    INIT := 100, // Initialisieren 
    Init_HomeVertical_10,
    Init_Vertical_10_Down,
    Init_HomeVertical_02,
    Init_Vertical_02_Up,
    Init_HomeHorizontal,
    Init_HorizontalToTrack,
    Init_check_if_pces_handled,

    READY := 999,  // READY to Start, Init Done 
    START := 1000, // Start Zyklisch

    waitOnMover,     // wait until the mover is there
    MOVER_NEEDED_OP, // Ab here, a mover in position is needed to perform the action

    lift_piece_and_down_to_pick,        // lift the piece with 180.10Z and go down simultaneously with 180.02Z
    close_griper_pick_piece,            // close the griper to pick the piece
    clamp_down_maintain_piece,          // the clamp (niederhalter) goes down and hold the piece in place
    take_out_piece_and_put_down_lifter, // 180.02Z goes up with the piece, 180.10Z goes down

    SYNC_MOVER_LEAVE, // MoverMan need to take the mover
    MOVER_FREE_OP,    // here, operation without mover can be done.

    hor_move_to_extraction_pipe, // 180.01Y move to the extraction pipe
    ver_down_in_pipe,            // 180.02Z move down to a secure position to release the piece
    open_griper_put_piece,
    clamp_up_to_rest_position,
    ver_up_empty, // 180.02z goes up without piece
    hor_to_track_pos,
    ver_down_waiting_for_mover, // go down again and wait until a mover is there

    DONE := 8000,  // Ablauf beendet 
    ERROR := 9000, // Fehler 
    _max
);
END_TYPE

(*
back to shuttle
check level NIO Box
*)

// ---- POUs/20_AUTO/ST180/ST180_Recipe_t.TcDUT
TYPE ST180_Recipe_t : 
STRUCT
    xUseVerLeft  : BOOL; // Is the left vertical picker element is used
    xUseVerRight : BOOL; // Is the right vertical picker element is used
END_STRUCT
END_TYPE

// ---- POUs/20_AUTO/ST185/ST185_Cylinders_e.TcTLEO
TYPE ST185_Cylinders_e :
(
    Greifer_Patrone_Links,
    Greifer_Patrone_Rechts,
    Niederhalter_Deckel_Links,
    Niederhalter_Deckel_Rechts
);
END_TYPE

// ---- POUs/20_AUTO/ST185/ST185_PnpHorPos_e.TcDUT
TYPE ST185_PnpHorPos_e : ST110_PnpHorPos_e;
END_TYPE

// ---- POUs/20_AUTO/ST185/ST185_PnpVerPos_e.TcDUT
TYPE ST185_PnpVerPos_e :
(
    up_waiting_mover,
    down_empty,
    up_full,
    down_full,
	up_after_unload,
    _max
);
END_TYPE

// ---- POUs/20_AUTO/ST185/ST185_Pnp_e.TcTLEO
{attribute 'qualified_only'}
{attribute 'strict'}
{attribute 'to_string'}
TYPE
ST185_Pnp_e :
(
    RESET := 0, // Reset

    INIT := 100, // Initialisieren 
    Init_HomeVertical_10,
    Init_Vertical_10_Down,
    Init_HomeVertical_02,
    Init_Vertical_02_Up,
    Init_HomeHorizontal,
    Init_HorizontalToTrack,
    Init_check_if_pces_handled,

    READY := 999,  // READY to Start, Init Done 
    START := 1000, // Start Zyklisch

    waitOnMover,     // wait until the mover is there
    MOVER_NEEDED_OP, // Ab here, a mover in position is needed to perform the action

    lift_piece_and_down_to_pick,        // lift the piece with 180.10Z and go down simultaneously with 180.02Z
    close_griper_pick_piece,            // close the griper to pick the piece
    clamp_down_maintain_piece,          // the clamp (niederhalter) goes down and hold the piece in place
    take_out_piece_and_put_down_lifter, // 180.02Z goes up with the piece, 180.10Z goes down

    SYNC_MOVER_LEAVE, // MoverMan need to take the mover
    MOVER_FREE_OP,    // here, operation without mover can be done.

    hor_move_to_extraction_pipe, // 180.01Y move to the extraction pipe
    ver_down_in_pipe,            // 180.02Z move down to a secure position to release the piece
    open_griper_put_piece,
    clamp_up_to_rest_position,
    ver_up_empty, // 180.02z goes up without piece
    hor_to_track_pos,
    ver_down_waiting_for_mover, // go down again and wait until a mover is there

    DONE := 8000,  // Ablauf beendet 
    ERROR := 9000, // Fehler 
    _max
);
END_TYPE

(*
back to shuttle
check level NIO Box
*)

// ---- POUs/20_AUTO/ST185/ST185_Recipe_t.TcDUT
TYPE ST185_Recipe_t : 
STRUCT
    xUseVerLeft  : BOOL; // Is the left vertical picker element is used
    xUseVerRight : BOOL; // Is the right vertical picker element is used
END_STRUCT
END_TYPE

// ---- POUs/20_AUTO/StationList_e.TcTLEO
// Only station with manual mode cylinders
{attribute 'qualified_only'}
TYPE StationList_e :
(
    ST105, // 0
    ST110, // 1
    ST115, // 2
    ST120, // 3
    ST125, // 4
    ST128, // 5
    ST130, // 6
    ST135, // 7
    ST140, // 8
    ST145, // 9
    ST150, // 10
    ST155, // 11
    ST160, // 12
    ST165, // 13
    ST170, // 14
    //ST174 // is ignored because it is a waiting station
    ST175, // 15
    ST176, // 16
    ST180, // 17
    ST185, // 18
	_max
);
END_TYPE

// ---- GVLs/AXIS.TcGVL
{attribute 'qualified_only'}
(*******************************************************************)
(* ACHSEN KONSTANTEN *)
(*******************************************************************)
VAR_GLOBAL CONSTANT

END_VAR
VAR_GLOBAL
    (*******************************************************************)
    (* ACHSEN Variablen *)
    (*******************************************************************)
    //Axis Allgemein Teachen und Anzeige
    bTeachAxisNr  : BYTE;                              // Zu Teachende Achse # (von HMI)
    bTeachInPos   : BYTE;                              // Achse in Position (Teachpos (99= nicht in Pos))
    bTeachPos     : ARRAY[0..Axis_e._max - 1] OF BYTE; // Achse Teach Position (Anzufahrende Position #)
    rTeachIncAxis : REAL := 0.1;                       // Axis Inching Wert
    rTeachVelo    : REAL := 10;                        // Achse Geschwindigkeit (Anzeige)
    rTeachPos     : REAL;                              // Achse Teach Position (Anzufahrende Position Wert)
    rTeachActPos  : REAL;                              // Achse AKTUELLE Position (AKTUEL
    rTeachPosMin  : REAL;                              // Achse PositionsminimumLER Position Wert)
    rTeachPosMax  : REAL;                              // Achse Positionsmaximum
    rJogVelo_pc   : REAL := REAL#10.0;                 // global jog velocity in pc

    btTeachArAxis : ARRAY[0..Axis_e._max - 1] OF ARRAY[0..8] OF structButton; (* Buttons AXIS
                                                    0: Disable 
                                                    1: Inching 
                                                    2: Slow 
                                                    3: Fast 
                                                    4: Move Abs/Rel   
                                                    5: Manu Move NEGATIVE
                                                    6: Manu Move POSITIVE  
													7: Start Homing 
													8: Teachpos Übernehmen*)
END_VAR

(*******************************************************************)
(* ACHSEN Positionen von HMI*)
(*******************************************************************)
VAR_GLOBAL RETAIN

END_VAR

// ---- GVLs/CONST.TcGVL
{attribute 'qualified_only' := ''}
VAR_GLOBAL CONSTANT
    (*******************************************************************)
    (* Globale KONSTANTEN *)
    (*******************************************************************)

    USE_SIMULATION  : BOOL := TRUE;
    BIND_WITH_TRACK : BOOL := TRUE;

    STATION_NUMBER           : INT   := 20;
    MAX_GROUP                : INT   := 6;
    MAX_STATION_PER_GROUP    : INT   := 8;
    MAX_RECIPE_NUMBER        : INT   := 11;
    MAX_TRACK_LENGTH         : LREAL := 10060;
    MAX_MOVER_SIZE           : LREAL := 200.0;
    MAX_VECTOR_LIST          : INT   := 10;
    MAX_CYLINDER_PER_STATION : INT   := 10;

END_VAR

// ---- GVLs/GVL.TcGVL
{attribute 'qualified_only'}
VAR_GLOBAL
    (*******************************************************************)
    (* Allgemeine Globale Variablen *)
    (*******************************************************************)
    (******* FREIGABEN *********)
    //ST01
    xFG_ST01akVZ : BOOL; // Vereinzelung Teil anwesend
    xFG_ST01akWT : BOOL; // WT anwesend
    //ST02
    xFG_ST02akWT : BOOL; // WT anwesend

    st105_aut : FB_AUT_105;    // Laden Filtergehäuse
    st110_aut : FB_AUT_110;    // Laden RFID-Ring
    st115_aut : FB_AUT_115;    // Laden kristal
    st120_aut : FB_AUT_120;    // Laden Solerohr
    st125_aut : FB_AUT_125;    // Laden filterhut
    st128_aut : FB_AUT_128;    // Control filterhut
    st130_aut : FB_AUT_130;    // Dosieren A
    st135_aut : FB_AUT_135;    // Dosieren B
    st140_aut : FB_AUT_140;    // Niveaukontrolle
    st145_aut : FB_AUT_145;    // Laden Patronendeckel
    st150_aut : FB_AUT_150;    // Utralson A
    st155_aut : FB_AUT_155;    // Ultrason B
    st160_aut : FB_AUT_160;    // Prüfig A
    st165_aut : FB_AUT_165;    // Prüfig B
    st170_aut : FB_AUT_170;    // Program RFID
    st175_aut : FB_AUT_175;    // Laser A
    st176_aut : FB_AUT_MODIFY; // Laser B
    st180_aut : FB_AUT_180;    // Entladen schlecht
    st185_aut : FB_AUT_185;    // Entladen gut
	
	ST130_01Y_Feedback_Offset : LREAL; // Offset automatically adjusted by ST140
	ST135_01Y_Feedback_Offset : LREAL; // Offset automatically adjusted by ST140

END_VAR

// ---- GVLs/HMI.TcGVL
{attribute 'qualified_only'}
VAR_GLOBAL
    (*******************************************************************)
    (* Globale HMI Variablen *)
    (*******************************************************************)
    xImmer0 : BOOL := FALSE; //ALLWAYS FALSE
    xImmer1 : BOOL := TRUE;  //ALLWAYS TRUE

    (*******************************************************************)
    (* Flags *)
    (*******************************************************************)
    enState   : enState; //SYSTEM STATUS
    xInitDone : BOOL;    //SYSTEM INITIALIZED
    xRefDone  : BOOL;    //Axis REF
    xAlarm    : BOOL;    //ALARM AKTIV
    xMessage  : BOOL;    //MELDUNG AKTIV
    xWait     : BOOL;    //ALLE FBs warten
    xAIRon    : BOOL;    //Luftdruck IO
    xSPC      : BOOL;    //SPC angewählt

    Tast_BL : BOOL; // ... 

    (*******************************************************************)
    (* Buttons *)
    (*******************************************************************)
    //Control
    btArMain : ARRAY[0..20] OF structButton; (*	
													0: AUTO
													1: STEP
													2: END
													3: MANU
													4: INIT
													5: STOP
													6: LEER
													7: QUIT
													8: RESET TEMP COUNTER
													9: START
													10: HUBTÜREn ALLE
													11: HUBTÜRE 1
													12: HUBTÜRE 2
													13: HUBTÜRE 3
													14: HUBTÜRE 4
												*)
    //Manual pneumatics
    // see below for button button instance 
    btManuCylinders : ARRAY[0..StationList_e._max] OF ARRAY[0..CONST.MAX_CYLINDER_PER_STATION] OF structButton;
    (* 
	 * [StationList_e.ST105] 0
     * [0]: Zyklus [1]: Robot get [2]: Robot set [3] Feeder
	 *
     * [StationList_e.ST110] 1
     * [0]: Zyklus [1]: Vacum Gripper left [2]: Vacum Gripper right [3]: Feeder
     *
     * [StationList_e.ST115] 2
     * [0]: Zyklus [1]: Gripper left [2]: Gripper right [3]: Feeder
     *
     * [StationList_e.ST120] 3
     * [0]: Zyklus [1]: Gripper left [2]: Gripper right [3]: Rotative cylinder left
     * [4]: Rotative cylinder right [5]: Hublader left [6]: Hublader right
	 * [7]: feeder left [8]: feeder right
     *
     * [StationList_e.ST125] 4
     * [0]: Zyklus [1]: Gripper left [2]: Gripper right [3]: lock cylinder left
     * [4]: lock cylinder right [5]: Gripper Solerohr left [6]: Gripper Solerohr right
	 * [7]: feeder 
     *
     * [StationList_e.ST130] 5
     * [0]: Zyklus [1]: cell open left [2]: cell open right [3]: cell fill left
     * [4]: cell fill right [5]: vib cell left [6]: vib cell right
	 * [7]: holder patrone [8]: vib patrone left [9]: vib patrone right [10]: Feeder 
     *
     * [StationList_e.ST135] 6
	 * dito ST130
	 *
     * [StationList_e.ST145] 8
     * [0]: Zyklus [1]: Vacum Gripper left [2]: Vacum Gripper right [3]: Feeder
	 *
     * [StationList_e.ST150] 9
     * [0]: Zyklus [1]: mover maintening [2]: start welding
	 *
     * [StationList_e.ST155] 10
     * [0]: Zyklus [1]: mover maintening [2]: start welding
	 *
     * [StationList_e.ST160] 11
     * [0]: Zyklus [1]: holder left [2]: holder right [3]: seal left
	 * [4]: seal right [5]: fill left [6]: fill right [7]: start test
	 *
     * [StationList_e.ST165] 12
     * [0]: Zyklus [1]: holder left [2]: holder right [3]: seal left
	 * [4]: seal right [5]: fill left [6]: fill right [7]: start test
	 *
     * [StationList_e.ST170] 13
     * [0]: Zyklus [1]: start test left [2]: start test right
	 *
     * [StationList_e.ST175] 14
     * [0]: Zyklus [1]: holder [2]: cabine in [3]: cabine out
	 * [4]: start laser
	 *
     * [StationList_e.ST180] 15
     * [0]: Zyklus [1]: Gripper left [2]: Gripper right 
	 * [3]: holder left [4]: holder right
	 *
     * [StationList_e.ST185] 11
     * [0]: Zyklus [1]:  [2]: 
     *)

    btArST150 : ARRAY[0..20] OF structButton; (*	0 : Start USS
	                                                1 : Reset US
											   *)

    btArForceCyclus     : ARRAY[0..StationList_e._max - 1] OF structButton;
    bArForceCyclusState : ARRAY[0..StationList_e._max - 1] OF BOOL;

    (*******************************************************************)
    (* ALARME  *)
    (*******************************************************************)
    strArALARM  : ARRAY[1..100] OF structAlarm;
    strArMSG    : ARRAY[1..100] OF structAlarm;
    xArAlarmHMI : ARRAY[1..9999] OF BOOL;

    (*******************************************************************)
    (* ANZEIGE - Werte *)
    (*******************************************************************)
    iSelectAxis     : LinearAxis_e := LinearAxis_e.ST110_01Y;
    iSelectAxisCopy : LinearAxis_e := LinearAxis_e._max;
    btCopyAxisCfg   : structButton;

    iSelectCylinder     : StationList_e := StationList_e.ST105;
    iSelectCylinderCopy : StationList_e := StationList_e._max;
    btCopyCylinderCfg   : structButton;

    iSelectJogAxis : Axis_e;

    (*******************************************************************)
    (* Cycle Time [STATION]*)
    (*******************************************************************)
    dwArStartTime_ms : ARRAY[0..StationList_e._max - 1] OF DWORD;
    dwArCycleTime_ms : ARRAY[0..StationList_e._max - 1] OF DWORD;

    lrPiecePerMinute : LREAL;

    PieceDoneTmp : DINT; // number of piece done since last reset

    (*******************************************************************)
    (* Recipe HMI management *)
    (*******************************************************************)
    btCopyRecipe  : structButton;
    btSetDefault  : structButton;
    movesNames    : ARRAY[0..LinearAxis_e._max - 1] OF ARRAY[0..CONST.MAX_VECTOR_LIST] OF STRING;
    cylinderNames : ARRAY[0..StationList_e._max - 1] OF ARRAY[0..CONST.MAX_CYLINDER_PER_STATION] OF STRING;

    (*******************************************************************)
    (* Mover manual bt *)
    (*******************************************************************)
    selectedShuttle : INT := 1; // selected shuttle from the HMI

    (*******************************************************************)
    (* Diverses *)
    (*******************************************************************)
    xWriteALlog : BOOL;         // Alarmlog schreiben in File
    btWritePers : structButton; // write pers data in filesystem

    sCurrentHMI2 : STRING; // ???
END_VAR

// ---- GVLs/IN.TcGVL
{attribute 'qualified_only'}
VAR_GLOBAL
    (*******************************************************************)
    (* EINGÄNGE Schrank A *)
    (*******************************************************************)
    (* Modul *)
    //-EL1809 16DI 155D2
    I000_                          AT %IX00.0 : BOOL; //
    I001_monitor_24V               AT %IX00.1 : BOOL; // Netzgerät Schaltschrank A Überwachung +24V
    I002_monitor_BR                AT %IX00.2 : BOOL; // Netzgerüt B&R Überwachung +24V
    I003_lufter_safety             AT %IX00.3 : BOOL; // Lüfter Safety ok
    I004_druckwachter_luftdruck_ok AT %IX00.4 : BOOL; // Druckwächter Luftdruck ok
    I005_klimagerat_ok             AT %IX00.5 : BOOL; // Klimagerät ok
    I006_                          AT %IX00.6 : BOOL; //
    I007_                          AT %IX00.7 : BOOL; //

    I010_distanzsensor_verschmutzung_140_51 AT %IX01.0 : BOOL; // Distanzsensor 140.51 Verschmutzung
    I011_distanzsensor_verschmutzung_140_52 AT %IX01.1 : BOOL; // Distanzsensor 140.52 Verschmutzung
    I012_                                   AT %IX01.2 : BOOL; // 
    I013_                                   AT %IX01.3 : BOOL; // 
    I014_                                   AT %IX01.4 : BOOL; // 
    I015_                                   AT %IX01.5 : BOOL; // 
    I016_                                   AT %IX01.6 : BOOL; // 
    I017_                                   AT %IX01.7 : BOOL; // 

    //-EL1809 16DI 155D7
    I020_ultraschall_bereit_150_20  AT %IX02.0 : BOOL; // Ultraschall 150.20 Bereit
    I021_ultraschall_fehler_150_20  AT %IX02.1 : BOOL; // Ultraschall 150.20 Fehler
    I022_ultraschall_us_on_150_20   AT %IX02.2 : BOOL; // Ultraschall 150.20 US on
    I023_ultraschall_nullpos_150_20 AT %IX02.3 : BOOL; // Ultraschall 150.20 Nullposition
    I024_ultraschall_bereit_155_20  AT %IX02.4 : BOOL; // Ultraschall 155.20 Bereit
    I025_ultraschall_fehler_155_20  AT %IX02.5 : BOOL; // Ultraschall 155.20 Fehler
    I026_ultraschall_us_on_155_20   AT %IX02.6 : BOOL; // Ultraschall 155.20 US on
    I027_ultraschall_nullpos_155_20 AT %IX02.7 : BOOL; // Ultraschall 155.20 Nullposifion

    I030_rfid_test_link_out1_170_20 AT %IX03.0 : BOOL; // RFID Test links 170.20 OUT 1
    I031_rfid_test_link_out2_170_20 AT %IX03.1 : BOOL; // RFID Test links 170.20 OUT 2
    I032_rfid_test_link_out3_170_20 AT %IX03.2 : BOOL; // RFID Test links 170.20 OUT 3
    I033_rfid_test_link_out1_170_21 AT %IX03.3 : BOOL; // RFID Test links 170.21 OUT 1
    I034_rfid_test_link_out2_170_21 AT %IX03.4 : BOOL; // RFID Test links 170.21 OUT 2
    I035_rfid_test_link_out3_170_21 AT %IX03.5 : BOOL; // RFID Test links 170.21 OUT 3
    I036_                           AT %IX03.6 : BOOL; // 
    I037_                           AT %IX03.7 : BOOL; // 

    //-EL1809 16DI 15602
    I040_ AT %IX04.0 : BOOL; // 
    I041_ AT %IX04.1 : BOOL; // 
    I042_ AT %IX04.2 : BOOL; // 
    I043_ AT %IX04.3 : BOOL; // 
    I044_ AT %IX04.4 : BOOL; // 
    I045_ AT %IX04.5 : BOOL; // 
    I046_ AT %IX04.6 : BOOL; // 
    I047_ AT %IX04.7 : BOOL; // 

    I050_ AT %IX05.0 : BOOL; // 
    I051_ AT %IX05.1 : BOOL; // 
    I052_ AT %IX05.2 : BOOL; // 
    I053_ AT %IX05.3 : BOOL; // 
    I054_ AT %IX05.4 : BOOL; // 
    I055_ AT %IX05.5 : BOOL; // 
    I056_ AT %IX05.6 : BOOL; // 
    I057_ AT %IX05.7 : BOOL; // 

    (*******************************************************************)
    (* EINGÄNGE Schrank B *)
    (*******************************************************************)
    (* Modul *)
    //-EL1809 16DI 10155D2
    I500_laser_sammelfehler_175          AT %IX50.0 : BOOL; // Sauger Laser 175.21 Sammelfehler
    I501_laser_filter_voll_175           AT %IX50.1 : BOOL; // Sauger Laser 175.21 Filter voll
    I502_laser_drehzahl_175              AT %IX50.2 : BOOL; // Sauger Laser 175.21 Drehzahl
    I503_laser_temperatur_175            AT %IX50.3 : BOOL; // Sauger Laser 175.21 Temperatur
    I504_distanzsensor_verschmutzung_125 AT %IX50.4 : BOOL; // Distanzsensor 125.51 Verschmutzung
    I505_uberwachung_24V                 AT %IX50.5 : BOOL; // Netzgerät Schaltschrank B Überwachung +24V
    I506_klimagerat_ok                   AT %IX50.6 : BOOL; // Klimagerät schaltschrank B ok
    I507_entladeBand_125_alarm           AT %IX50.7 : BOOL; // Entladeband 185.21 Alarm

    I510_lufter_safey_ok AT %IX51.0 : BOOL; // Lüfter Safety Schaltschrank B ok
    I511_                AT %IX51.1 : BOOL; // 
    I512_                AT %IX51.2 : BOOL; // 
    I513_                AT %IX51.3 : BOOL; // 
    I514_                AT %IX51.4 : BOOL; // 
    I515_                AT %IX51.5 : BOOL; // 
    I516_                AT %IX51.6 : BOOL; // 
    I517_                AT %IX51.7 : BOOL; // 

    //-EL1809 16DI 1015507
    I520_                AT %IX52.0 : BOOL; // 
    I521_ AT %IX52.1 : BOOL; // 
    I522_                AT %IX52.2 : BOOL; // 
    I523_ AT %IX52.3 : BOOL; // 
    I524_                AT %IX52.4 : BOOL; // 
    I525_ AT %IX52.5 : BOOL; // 
    I526_                AT %IX52.6 : BOOL; // 
    I527_ AT %IX52.7 : BOOL; // 

    I530_ AT %IX53.0 : BOOL; // 
    I531_ AT %IX53.1 : BOOL; // 
    I532_ AT %IX53.2 : BOOL; // 
    I533_ AT %IX53.3 : BOOL; // 
    I534_ AT %IX53.4 : BOOL; // 
    I535_ AT %IX53.5 : BOOL; // 
    I536_ AT %IX53.6 : BOOL; // 
    I537_ AT %IX53.7 : BOOL; // 

    AI01_ST140_level_track_side AT %I* : UINT; // laser sensor used to measure powder level, placed at the track side
    AI02_ST140_level_door_side  AT %I* : UINT; // laser sensor used to measure powder level, placed at the door side

    AI11_ST130_valve_feedback_left  AT %I* : UINT; // current flow of the proportional valve
    AI12_ST130_valve_feedback_right AT %I* : UINT; // current flow of the proportional valve
    AI13_ST135_valve_feedback_left  AT %I* : UINT; // current flow of the proportional valve
    AI14_ST135_valve_feedback_right AT %I* : UINT; // current flow of the proportional valve

    AI21_ST125_piece_height AT %I* : UINT; // laser sensor value, detect pieces in round table
    AI22_                   AT %I* : UINT;

    I_CPX9_1_ResetBp AT %I* : BOOL; // Blue button on the panel
    I_CPX9_1_greenBp AT %I* : BOOL; // Green button on the panel
    I_CPX9_1_redBp   AT %I* : BOOL; // Red button on the panel

END_VAR

// ---- GVLs/IO_BOX.TcGVL
{attribute 'qualified_only'}
VAR_GLOBAL
    (*******************************************************************)
    (* EINGÄNGE Schrank A *)
    (*******************************************************************)

    (* IO-Link Boxen 190A1 *)
    (*******************************************************************)
    //-194A3
    (* BN Lampe *)
    I0000_ AT %Q* : BOOL; // lampe

    //-201A1
    (* Ventil Batterie 201 A*)
    Q0100_14_ST130_kammer_offnen_links     AT %Q* : BOOL; // ST130 Kammer öffnen links
    Q0100_12_                              AT %Q* : BOOL; // 
    Q0101_14_ST130_kammer_offnen_rechts     AT %Q* : BOOL; // ST130 Kammer öffnen rechts
    Q0101_12_                              AT %Q* : BOOL; // 
    Q0102_14_ST130_kammer_nachfullen_links  AT %Q* : BOOL; // ST130 Kammer nachfüllen links
    Q0102_12_                              AT %Q* : BOOL; // 
    Q0103_14_ST130_kammer_nachfullen_rechts AT %Q* : BOOL; // ST130 Kammer nachfüllen rechts
    Q0103_12_                              AT %Q* : BOOL; // 
    Q0104_14_ST130_vibrieren_kammer_links   AT %Q* : BOOL; // ST130 Vibrieren Kammer links/rechts aus
    Q0104_12_ST130_vibrieren_kammer_rechts AT %Q* : BOOL; // ST130 Vibrieren Kammer links/rechts ein
    Q0105_14_ST130_niederhalter_patrone    AT %Q* : BOOL; // ST130 Niederhalter Patrone
    Q0105_12_                              AT %Q* : BOOL; // 
    Q0106_14_ST135_kammer_offnen_links      AT %Q* : BOOL; // ST135 Kammer öffnen links
    Q0106_12_                              AT %Q* : BOOL; // 
    Q0107_14_ST135_kammer_offnen_rechts     AT %Q* : BOOL; // ST135 Kammer öffnen rechts
    Q0107_12_                              AT %Q* : BOOL; // 
    Q0108_14_ST135_kammer_nachfullen_links  AT %Q* : BOOL; // ST135 Kammer nachfüllen links
    Q0108_12_                              AT %Q* : BOOL; // 
    Q0109_14_ST135_kammer_nachfullen_rechts AT %Q* : BOOL; // ST135 Kammer nachfüllen rechts
    Q0109_12_                              AT %Q* : BOOL; // 
    Q0110_14_ST135_vibrieren_kammer_links   AT %Q* : BOOL; // ST135 Vibrieren Kammer links 
    Q0110_12_ST135_vibrieren_kammer_rechts AT %Q* : BOOL; // ST135 Vibrieren Kammer rechts
    Q0111_14_ST135_niederhalter_patrone    AT %Q* : BOOL; // ST135 Niederhalter Patrone
    Q0111_12                               AT %Q* : BOOL; //
    Q0112_14_                               AT %Q* : BOOL; //
    Q0112_12_                              AT %Q* : BOOL; // 
    Q0113_14_                               AT %Q* : BOOL; //
    Q0113_12_                              AT %Q* : BOOL; // 
    Q0114_14_                               AT %Q* : BOOL; //
    Q0114_12_                              AT %Q* : BOOL; // 
    Q0115_14_                               AT %Q* : BOOL; //
    Q0115_12_                              AT %Q* : BOOL; // 

    //-202A1
    (* Ventil Batterie 202 A *)
    Q0200_14_ST145_vakum_greifer_links  AT %Q* : BOOL; // 
    Q0200_12_                           AT %Q* : BOOL; // Vakumgreifer links ST145
    Q0201_14_ST145_vakum_greifer_rechts AT %Q* : BOOL; // 
    Q0201_12_                           AT %Q* : BOOL; // Vakumgreifer rechts ST145
    Q0202_14_ST150_kraftubersetzung     AT %Q* : BOOL; // 
    Q0202_12_                           AT %Q* : BOOL; // Kraftübersetzung ST150
    Q0203_14_ST155_kraftubersetzung     AT %Q* : BOOL; // 
    Q0203_12_                           AT %Q* : BOOL; // Kraftübersetzung ST155
    Q0204_14_                           AT %Q* : BOOL; // 
    Q0204_12_                           AT %Q* : BOOL; // 
    Q0205_14_                           AT %Q* : BOOL; // 
    Q0205_12_                           AT %Q* : BOOL; // 

    //-203A1
    (* Ventil Batterie 203 A *)
    Q0300_14_ST160_niederhalter_links         AT %Q* : BOOL; // ST160 Niederhalter links ST160
    Q0300_12_                                 AT %Q* : BOOL; // 
    Q0301_14_ST160_niederhalter_rechts        AT %Q* : BOOL; // ST160 Niederhalter rechts ST160
    Q0301_12_                                 AT %Q* : BOOL; // 
    Q0302_14_ST160_dichtung_pruflocker_links  AT %Q* : BOOL; // ST160 Dichtung Prüfglocker links
    Q0302_12_ST160_dichtung_pruflocker_rechts AT %Q* : BOOL; // ST160 Dichtung Prüfglocker rechts
    Q0303_14_nc                               AT %Q* : BOOL; // ST160 not connected (yet?)
    Q0303_12_nc                               AT %Q* : BOOL; // ST160 not connected (yet?)
    Q0304_14_ST165_niederhalter_links         AT %Q* : BOOL; // ST165 Niederhalter links ST160   
    Q0304_12_                                 AT %Q* : BOOL; //                                  
    Q0305_14_ST165_niederhalter_rechts        AT %Q* : BOOL; // ST165 Niederhalter rechts ST160  
    Q0305_12_                                 AT %Q* : BOOL; // 
    Q0306_14_ST165_dichtung_pruflocker_links  AT %Q* : BOOL; // ST165 Dichtung Prüfglocker links 
    Q0306_12_ST165_dichtung_pruflocker_rechts AT %Q* : BOOL; // ST165 Dichtung Prüfglocker rechts
    Q0307_14_nc                               AT %Q* : BOOL; // ST165 not connected (yet?)       
    Q0307_12_nc                               AT %Q* : BOOL; // ST165 not connected (yet?)       
    Q0308_14_                                 AT %Q* : BOOL; // 
    Q0308_12_                                 AT %Q* : BOOL; // 
    Q0309_14_                                 AT %Q* : BOOL; // 
    Q0309_12_                                 AT %Q* : BOOL; // 
    Q0310_14_                                 AT %Q* : BOOL; // 
    Q0310_12_                                 AT %Q* : BOOL; // 
    Q0311_14_                                 AT %Q* : BOOL; // 
    Q0311_12_                                 AT %Q* : BOOL; // 

    (* IO-Link Boxen 190A4 *)
    (*******************************************************************)
    //-970B2
    (* FullstandKontrolle ST130.55 *)
    I1000_ AT %I* : BOOL; // FullstandKontrolle ST130.55

    //-970B4
    (* FullstandKontrolle ST130.56 *)
    I1100_ AT %I* : BOOL; // FullstandKontrolle ST130.56

    //-970B6
    (* FullstandKontrolle ST135.55 *)
    I1200_ AT %I* : BOOL; // FullstandKontrolle ST135.55

    //-970B7
    (* FullstandKontrolle ST135.56 *)
    I1300_ AT %I* : BOOL; // 

    //-5009
    (* ST130 I - 8x IO *)
    I1400_ST130_nachfullen_offnen_links_zuruck  AT %I* : BOOL; // 0: Kammer öffnen links zurück
    I1401_ST130_nachfullen_offnen_links_vor     AT %I* : BOOL; // 1: Kammer öffnen links vor
    I1402_ST130_nachfullen_offnen_rechts_zuruck AT %I* : BOOL; // 2: Kammer öffnen rechts zurück
    I1403_ST130_nachfullen_offnen_rechts_vor    AT %I* : BOOL; // 3: Kammer öffnen rechts vor
    I1404_ST130_kammer_offnen_links_zuruck      AT %I* : BOOL; // 4: Kummer nachfüllen links zurück
    I1405_ST130_kammer_offnen_links_vor         AT %I* : BOOL; // 5: Kummer nachfüllen links vor
    I1406_ST130_kammer_offnen_rechts_zuruck     AT %I* : BOOL; // 6: Kammer nachfüllen rechts zurück
    I1407_ST130_kammer_offnen_rechts_vor        AT %I* : BOOL; // 7: Kammer nachfüllen rechts vor

    //-5010
    (* ST135 I - 8x IO *)
    I1500_ST135_nachfullen_offnen_links_zuruck AT %I* : BOOL; // 0: Kammer öffnen links zurück
    I1501_ST135_nachfullen_offnen_rechts_vor   AT %I* : BOOL; // 1: Kammer öffnen links vor
    I1502_ST135_nachfullen_offnen_links_zuruck AT %I* : BOOL; // 2: Kammer öffnen rechts zurück
    I1503_ST135_nachfullen_offnen_rechts_vor   AT %I* : BOOL; // 3: Kammer öffnen rechts vor
    I1504_ST135_kammer_offnen_links_zuruck     AT %I* : BOOL; // 4: Kummer nachfüllen links zurück
    I1505_ST135_kammer_offnen_rechts_vor       AT %I* : BOOL; // 5: Kummer nachfüllen links vor
    I1506_ST135_kammer_offnen_links_zuruck     AT %I* : BOOL; // 6: Kammer nachfüllen rechts zurück
    I1507_ST135_kammer_offnen_rechts_vor       AT %I* : BOOL; // 7: Kammer nachfüllen rechts vor

    //-5014
    (* ST145 I - 4x IO *)
    I1600_ST145_vakum_teil_in_greiffer_left  AT %I* : BOOL; // 0: Vakuumkontrolle Teil in Greifer 145.03
    I1601_ST145_vakum_teil_in_greiffer_right AT %I* : BOOL; // 1: Vakuumkontrolle Teil in Greifer 145.04

    (* IO-Link Boxen 190A8 *)
    (*******************************************************************)
    //-5011
    (* Filterhut vorhanden ST130/135 I - 8x IO *)
    I2000_ST128_filterhut_vorhanden AT %I* : BOOL; // 0: ST130 Filterhut vorhanden links
    //
    I2001_ AT %I* : BOOL; // 
    I2002_ AT %I* : BOOL; // 
    I2003_ AT %I* : BOOL; // 
    I2004_ AT %I* : BOOL; // 
    I2005_ AT %I* : BOOL; // 
    I2006_ AT %I* : BOOL; // 
    I2007_ AT %I* : BOOL; // 

    //-5012
    (* Niederhalter Patrone ST130/135 I - 8x IO *)
    I2100_ST130_niederhalter_patrone_oben  AT %I* : BOOL; // 0: ST130 Niederhalter Patrone oben
    I2101_ST130_niederhalter_patrone_unten AT %I* : BOOL; // 1: ST130 Niederhalter Patrone unten
    I2102_ST135_niederhalter_patrone_oben  AT %I* : BOOL; // 2: ST135 Niederhalter Patrone oben
    I2103_ST135_niederhalter_patrone_unten AT %I* : BOOL; // 3: ST135 Niederhalter Patrone unten

    //-5013
    (* Niederhalter & Vorsatzwanne ST130 I - 8x IO *)
    I2200_ST130_niederhalter_vorne  AT %I* : BOOL; // 0: Niederhalter in Arbeitspos. vorne
    I2201_ST130_niederhalter_hinten AT %I* : BOOL; // 1: Niederhalter in Wartungspos. hinten
    I2202_ST130_Vorsatzwanne_vorne  AT %I* : BOOL; // 2: Vorsatzwanne in Arbeitspos. vorne
    I2203_ST130_Vorsatzwanne_hinten AT %I* : BOOL; // 3: Vorsatzwanne in Ruhepos. hinten

    //-5015
    (* ST145/150/155 I - 8x IO *)
    I2300_ST145_teil_in_vereinzelung    AT %I* : BOOL; // 0: AWK Teil in Vereinzelung (RST) ST145
    I2301_ST150_kraftubersetzung_zuruck AT %I* : BOOL; // 1: Kraftübersetzung zurück ST150
    I2302_ST150_kraftubersetzung_vor    AT %I* : BOOL; // 2: Kraftübersetzung vor ST150
    I2303_ST150_deckel_vohanden         AT %I* : BOOL; // 3: Deckel vorhanden ST150
    I2304_ST155_kraftubersetzung_zuruck AT %I* : BOOL; // 4: Kraftübersetzung zurück ST155
    I2305_ST155_kraftubersetzung_vor    AT %I* : BOOL; // 5: Kraftübersetzung vor ST155
    I2306_ST155_deckel_vohanden         AT %I* : BOOL; // 6: Deckel vorhanden ST155

    //-5501
    (* feeder ST145 *)
    Q2400_ST145_freigabe_REO AT %Q* : BOOL; // 0: Freigabe REO
    I2401_ST145_maximum_wf   AT %I* : BOOL; // 1: Maximum WF
    Q2402_ST145_reigabe_wf   AT %Q* : BOOL; // 2: Freigabe WF

    (* IO-Link Boxen 191A2 *)
    (*******************************************************************)
    //-960B2
    (* Wegmessenor ST160.02 *)
    I3000_ST160_Wegmessenor_links AT %I* : UINT;

    //-960B4
    (* Wegmessenor ST160.03 *)
    I3100_ST160_Wegmessenor_rechts AT %I* : UINT;

    //-960B6
    (* Wegmessenor ST165.02 *)
    I3200_ST165_Wegmessenor_links AT %I* : UINT;

    //-960B7
    (* Wegmessenor ST165.03 *)
    I3300_ST165_Wegmessenor_rechts AT %I* : UINT;

    (*******************************************************************)
    (* EINGÄNGE Schrank B *)
    (*******************************************************************)

    (* IO-Link Boxen 1012045.1 *)
    (*******************************************************************)
    //-10194A3
    (* Meldeleuchte 3 Zonen mit Horni BNI0086 *)
    Q5000_ : BOOL; // eldeleuchte 3 Zonen mit Horni BNI0086

    //-10201B1
    (* Ventilbat. 201 B *)
    // empty
    //Q5100_ AT %Q* : BOOL; // eldeleuchte 3 Zonen mit Horni BNI0086

    //-10202B1
    (* Ventilbat. 202 B - 16 slots *)
    Q5200_14_ST115_greifer_links AT %Q* : BOOL; // Greifer links ST115           
    Q5200_12_                    AT %Q* : BOOL; //                               
    Q5201_14_ST115_greifer_rechts           AT %Q* : BOOL; // Greifer rechts ST115          
    Q5201_12_                    AT %Q* : BOOL; //                               
    Q5202_14_ST120_greifer_links            AT %Q* : BOOL; // Greifer links ST120           
    Q5202_12_                    AT %Q* : BOOL; //                               
    Q5203_14_ST120_greifer_rechts           AT %Q* : BOOL; // Greifer rechts ST120          
    Q5203_12_                    AT %Q* : BOOL; //                               
    Q5204_14_ST120_schwenken_links          AT %Q* : BOOL; // Schwenken links ST120         
    Q5204_12_                    AT %Q* : BOOL; //                               
    Q5205_14_ST120_schwenken_rechts         AT %Q* : BOOL; // Schwenken rechts ST120        
    Q5205_12_                    AT %Q* : BOOL; //                               
    Q5206_14_ST125_greifer_filterhut_links  AT %Q* : BOOL; // Greifer Filterhut links ST125 
    Q5206_12_                    AT %Q* : BOOL; //                               
    Q5207_14_ST125_greifer_filterhut_rechts AT %Q* : BOOL; // Greifer Filterhut rechts ST125
    Q5207_12_                    AT %Q* : BOOL; //                               
    Q5208_14_ST125_handling_solerohr_links  AT %Q* : BOOL; // Handling Solerohr links ST125 
    Q5208_12_                    AT %Q* : BOOL; //                               
    Q5209_14_ST125_handling_solerohr_rechts AT %Q* : BOOL; // Handling Solerohr rechts ST125
    Q5209_12_                    AT %Q* : BOOL; //                               
    Q5210_14_ST125_greifer_solerohr_links   AT %Q* : BOOL; // Greifer Solerohr links ST125  
    Q5210_12_                    AT %Q* : BOOL; //                               
    Q5211_14_ST125_greifer_solerohr_rechts  AT %Q* : BOOL; // Greifer Solerohr rechts ST125 
    Q5211_12_                    AT %Q* : BOOL; //                               
    Q5212_14_ST120_stop_vertical_axis AT %Q* : BOOL; // 
    Q5212_12_                    AT %Q* : BOOL; // 
    Q5213_14_                               AT %Q* : BOOL; // 
    Q5213_12_                    AT %Q* : BOOL; // 
    Q5214_14_                               AT %Q* : BOOL; // 
    Q5214_12_                    AT %Q* : BOOL; // 
    Q5215_14_                               AT %Q* : BOOL; // 
    Q5215_12_                    AT %Q* : BOOL; // 

    //-10203B1
    (* Ventilbat. 203 B - 5 slots *)
    Q5300_14_ST175_niederhalter AT %Q* : BOOL; // q0: Niederhalter ST175     
    Q5300_12_                   AT %Q* : BOOL; //                            
    Q5301_14_ST175_kabinentur_einlaufseite AT %Q* : BOOL; // q1: Kabinentür Einlaufseite
    Q5301_12_                   AT %Q* : BOOL; //                            
    Q5302_14_ST175_kabinentur_auflaufseite AT %Q* : BOOL; // q2: Kabinentür Auflaufseite
    Q5302_12_                   AT %Q* : BOOL; //                            
    Q5303_14_                              AT %Q* : BOOL; // q3:                        
    Q5303_12_                   AT %Q* : BOOL; //                            
    Q5304_14_                              AT %Q* : BOOL; // q4:                        
    Q5304_12_                   AT %Q* : BOOL; // 

    //-10204B1
    (* Ventilbat. 204 B - 12 slots *)
    Q5400_14_ST180_greifer_patrone_links AT %Q* : BOOL; // Greifer Patrone links ST180     
    Q5400_12_                            AT %Q* : BOOL; //                                 
    Q5401_14_ST180_greifer_patrone_rechts     AT %Q* : BOOL; // Grefier Patrone rechts ST180    
    Q5401_12_                            AT %Q* : BOOL; //                                 
    Q5402_14_ST180_niederhalter_deckel_links  AT %Q* : BOOL; // Niederhalter Deckel links ST180 
    Q5402_12_                            AT %Q* : BOOL; //                                 
    Q5403_14_ST180_Niederhalter_deckel_rechts AT %Q* : BOOL; // Niederhalter Deckel rechts ST180
    Q5403_12_                            AT %Q* : BOOL; //                                 
    Q5404_14_ST185_greifer_patrone_links      AT %Q* : BOOL; // Greifer Patrone links ST185     
    Q5404_12_                            AT %Q* : BOOL; //                                 
    Q5405_14_ST185_greifer_patrone_rechts     AT %Q* : BOOL; // Greifer Patrone rechts ST185    
    Q5405_12_                            AT %Q* : BOOL; //                                 
    Q5406_14_ST185_niederhalter_deckel_links  AT %Q* : BOOL; // Niederhalter Deckel links ST185 
    Q5406_12_                            AT %Q* : BOOL; //                                 
    Q5407_14_ST185_Niederhalter_deckel_rechts AT %Q* : BOOL; // Niederhalter Deckel rechts ST185
    Q5407_12_                            AT %Q* : BOOL; //                                 
    Q5408_14_ST180_Break_axis_02Z AT %Q* : BOOL; //                                 
    Q5408_12_                            AT %Q* : BOOL; //                                 
    Q5409_14_ST185_Break_axis_02Z AT %Q* : BOOL; //                                 
    Q5409_12_                            AT %Q* : BOOL; // 
    Q5410_14_                                 AT %Q* : BOOL; // 
    Q5410_12_                            AT %Q* : BOOL; // 
    Q5411_14_                                 AT %Q* : BOOL; // 
    Q5411_12_                            AT %Q* : BOOL; // 

    //-10950B1
    (* Vakuumsch. Greifer 110.05 *)
    I5500_ST110_vakumkontrolle_links AT %I* : INT; // Vakuumsch. Greifer 110.05

    //-10950B3
    (* Vakuumsch. Greifer 110.06 *)
    I5600_ST110_vakumkontrolle_rechts AT %I* : INT; // Vakuumsch. Greifer 110.05

    (* IO-Link Boxen 10120A5.2 *)
    (*******************************************************************)
    //-5002
    (* Teil in Vereinzelung (RST) ST110/115 - 8x IO *)
    I6000_ST110_teil_in_vereinzelung AT %I* : BOOL; // Teil in Vereinzelung (RST) ST110
    I6001_ST115_teil_in_vereinzelung AT %I* : BOOL; // Teil in Vereinzelung (RST) ST115

    //-5003
    (* Greifer links ST115 - 4x IO *)
    I6100_ST115_greifer_links_offen       AT %I* : BOOL; // 0: Greifer links offen
    I6101_ST115_greifer_links_geschlossen AT %I* : BOOL; // 1: Greifer links geschlossen

    //-5004
    (* Greifer recht ST115 - 4x IO  *)
    I6200_ST115_greifer_rechts_offen       AT %I* : BOOL; // 0: Greifer rechts offen
    I6201_ST115_greifer_rechts_geschlossen AT %I* : BOOL; // 1: Greifer rechts geschlossen

    //-5005
    (* Greifern link & rechts ST120 - 4x IO*)
    I6300_ST120_greifer_links_geschlossen  AT %I* : BOOL; // 0: Greifer links geschlossen
    I6301_ST120_greifer_links_offen        AT %I* : BOOL; // 1: Greifer links offen
    I6302_ST120_greifer_rechts_geschlossen AT %I* : BOOL; // 2: Greifer rechts geschlossen
    I6303_ST120_greifer_rechts_offen       AT %I* : BOOL; // 3: Greifer rechts offen

    //-5006
    (* feeder ST120 - 8x IO *)
    I6400_ST120_schwenken_links_in_vertikal    AT %I* : BOOL; // 0: Schwenken links vertikal
    I6401_ST120_schwenken_links_in_horizontal  AT %I* : BOOL; // 1: Schwenken links horizontal
    I6402_ST120_schwenken_rechts_in_vertikal   AT %I* : BOOL; // 2: Schwenken rechts vertikal
    I6403_ST120_schwenken_rechts_in_horizontal AT %I* : BOOL; // 3: Schwenken rechts horizontal
    I6404_ST120_teil_in_vereizelung_links      AT %I* : BOOL; // 4: Teil in Vereinzelung links
    I6405_ST120_teil_in_vereinzelung_rechts    AT %I* : BOOL; // 5: Teil in Vereinzelung rechts

    //-5007
    (* Pnp Filterhut Greifer ST125 - 4x IO*)
    I6500_ST125_greiffer_filterhut_links_geschlossen  AT %I* : BOOL; // 0: G. Filterhut links geschlossen
    I6501_ST125_greiffer_filterhut_links_offen        AT %I* : BOOL; // 1: G. Filterhut links offen
    I6502_ST125_greiffer_filterhut_rechts_geschlossen AT %I* : BOOL; // 2: G. Filterhut rechts geschlossen
    I6503_ST125_greiffer_filterhut_rechts_offen       AT %I* : BOOL; // 3: G. Filterhut rechts offen

    //-5008
    (* Pnp Solerohr Greiffer ST125 - 8x IO *)
    I6600_ST125_solerhor_handling_links_unten       AT %I* : BOOL; // 0: Solerohr handling links unten
    I6601_ST125_solerhor_handling_links_oben        AT %I* : BOOL; // 1: Solerohr handling links oben
    I6602_ST125_solerhor_handling_rechts_unten      AT %I* : BOOL; // 2: Solerohr handling rechts unten
    I6603_ST125_solerhor_handling_rechts_oben       AT %I* : BOOL; // 3: Solerohr handling rechts oben
    I6604_ST125_greifer_solerohr_links_geschlossen  AT %I* : BOOL; // 4: G.Solerohr links geschlossen
    I6605_ST125_greifer_solerohr_links_offen        AT %I* : BOOL; // 5: G.Solerohr links offen
    I6606_ST125_greifer_solerohr_rechts_geschlossen AT %I* : BOOL; // 6: G.Solerohr rechts geschlossen
    I6607_ST125_greifer_solerohr_rechts_offen       AT %I* : BOOL; // 7: G.Solerohr rechts offen

    (* IO-Link Boxen 10190A8 *)
    (*******************************************************************)
    //-10945.2 / 110.55
    (* Wandler Kraftsensor 110 links *)
    I7000_ST110_kraftsensor_links AT %I* : BOOL;

    //-10945.3 / 110.56
    (* Wandler Kraftsensor 110 rechts *)
    I7100_ST110_kraftsensor_rechts AT %I* : BOOL;

    //-10945.3 / 115.55
    (* Wandler Kraftsensor 115 links *)
    I7200_ST115_kraftsensor_links AT %I* : BOOL;

    //-10945.5 / 115.56
    (* Wandler Kraftsensor 115 rechts *)
    I7300_ST115_kraftsensor_rechts AT %I* : BOOL;

    //-10945.7 / 120.55
    (* Wandler Kraftsensor 120 links *)
    I7400_ST120_kraftsensor_links AT %I* : BOOL;

    //-10945.8 / 120.56
    (* Wandler Kraftsensor 120 rechts *)
    I7500_ST120_kraftsensor_rechts AT %I* : BOOL;

    //-10946.2 / 125.55
    (* Wandler Kraftsensor 125 links *)
    I7600_ST125_kraftsensor_links AT %I* : BOOL;

    //-10946.3 / 125.56
    (* Wandler Kraftsensor 125 rechts *)
    I7700_ST125_kraftsensor_rechts AT %I* : BOOL;

    (* IO-Link Boxen 10191A2 *)
    (*******************************************************************)
    //-15501
    (* feeder ST110 - 8x IO *)
    Q8000_ST110_freigabe_wf              AT %Q* : BOOL; // 0: Freigabe WF ST110
    I8001_ST110_maximum                  AT %I* : BOOL; // 1: Maximum WF ST110
    I8002_ST110_alarm_forderband         AT %I* : BOOL; // 2: Alarm Förderband ST110
    Q8003_ST110_forderband_ein           AT %Q* : BOOL; // q3: Förderband ein ST110
    I8004_ST110_farbsensor_lagekontrolle AT %I* : BOOL; // 4: Farbsensor Lagekontrolle
    Q8005_ST110_blow_piece               AT %Q* : BOOL; // q5: blow top black pieces into the feeder

    //-15502
    (* feeder ST115 - 8x IO *)
    Q8100_ST115_freigabe_wf      AT %Q* : BOOL; // q0: Freigabe WF ST115
    I8101_ST115_maximum          AT %I* : BOOL; // 1: Maximum WF ST115
    I8102_ST115_alarm_forderband AT %I* : BOOL; // 2: Alarm Förderband ST115
    Q8103_ST115_forderband_ein   AT %Q* : BOOL; // q3: Förderband ein ST115

    //-15503
    (* feeder links ST120 - 8x IO *)
    I8200_ST120_alarm_forderband_l             AT %I* : BOOL; //  0: Alarm Förderband ST115
    Q8201_ST120_forderband_ein_l               AT %Q* : BOOL; // q1: Förderband ein
    I8202_ST120_alarm_forderband_r             AT %I* : BOOL; //  2: Alarm Förderband
    Q8203_ST120_forderband_ein_r               AT %Q* : BOOL; // q3: Förderband ein
    I8204_ST120_hublader_links_unten           AT %I* : BOOL; //  4: Hublader links unten
    I8205_ST120_hublader_links_oben            AT %I* : BOOL; //  5: Hublader links oben
    I8206_ST120_hublader_links_niveaukontrolle AT %I* : BOOL; //  6: Hublader links Nivaukontrolle
    Q8207_ST120_hublader_links_valve           AT %Q* : BOOL; // q7: Hublader links 120.12

    //-15504
    (* feeder rechts ST120 - 8x IO *)
    I8300_ST120_hublader_rechts_unten           AT %I* : BOOL; //  0: Hublader rechts unten
    I8301_ST120_hublader_rechts_oben            AT %I* : BOOL; //  1: Hublader rechts oben
    I8302_ST120_hublader_rechts_niveaukontrolle AT %I* : BOOL; //  2: Hublader rechts Nivaukontrolle
    Q8303_ST120_hublader_rechts_valve           AT %Q* : BOOL; // q3: Hublader rechts 120.13
    I8304_ST120_maxi_zufurung_links             AT %I* : BOOL; //  4: Mini-Maxi Kontrolle Zuführung links
    I8305_ST120_maxi_zufurung_rechts            AT %I* : BOOL; //  5: Mini-Maxi Kontrolle Zuführung rechts

    //-15505
    (* feeder ST125 - 8x IO *)
    Q8400_ST125_freigabe_REO AT %Q* : BOOL; // q0: Freigabe REO
    I8401_ST125_maximum_wf   AT %I* : BOOL; //  1: Maximum WF
    Q8402_ST125_freigabe_wf  AT %Q* : BOOL; // q2: Freigabe WF

    //-5001
    (* feeder ST105 and ST101 - 8x I *)
    I8600_ST105_teil_in_vereinzelung     AT %I* : BOOL; // 1: Teil in Vereinzelung (RST)
    I8601_ST105_shuttle_pin_config_pro   AT %I* : BOOL; // 2: Kontrolle WT-Hülsen Typ Pro
    I8602_ST105_shuttle_pin_config_maxi  AT %I* : BOOL; // 3: Kontrolle WT- Schieber verriegelt
    I8603_ST105_shuttle_ring_pro_present AT %I* : BOOL; // 4: Kontrolle WT- Schieber entriegelt
    I8604_ST105_first_shuttle_pin        AT %I* : BOOL; // 5: Anwesenheit, Init. WT Nr.1

    //-15500
    (* feeder ST105 - 8x IO *)
    I8700_ST105_Ausheber_unten_GS             AT %I* : BOOL; // 1: 
    I8701_ST105_Ausheber_oben_AS              AT %I* : BOOL; // 2: 
    I8702_ST105_Abschieber_zuruck_GS          AT %I* : BOOL; // 3: 
    I8703_ST105_Abschieber_vor_AS             AT %I* : BOOL; // 4: 
    I8704_ST105_Maximum_LF                    AT %I* : BOOL; // 5: 
    I8705_ST105_Kontrolle_zwei_Filtergehiluse AT %I* : BOOL; // 6: 
    I8706_ST105_                              AT %I* : BOOL; // 7: 
    I8707_ST105_                              AT %I* : BOOL; // 8: 

    //-10201B1
    (* Ventilbat. 204 B - 12 slots *)
    Q8800_14_Auschieber_ab_auf     AT %Q* : BOOL; //
	Q8800_12_ AT %Q* : BOOL; // 
    Q8801_14_Auschieber_vor_zuruck AT %Q* : BOOL; // 
	Q8801_12_ AT %Q* : BOOL; // 
    Q8802_14_                      AT %Q* : BOOL; // 
	Q8802_12_ AT %Q* : BOOL; // 
    Q8803_14_                      AT %Q* : BOOL; // 
	Q8803_12_ AT %Q* : BOOL; // 
    Q8804_14_                      AT %Q* : BOOL; // 
	Q8804_12_ AT %Q* : BOOL; // 
    Q8805_14_                      AT %Q* : BOOL; // 
	Q8805_12_ AT %Q* : BOOL; // 

    (* IO-Link Boxen 10191A5 *)
    (*******************************************************************)
    //-5016
    (* ST175/180 8x IO *)
    I9000_ST175_kabinentur_einlauf_offen      AT %I* : BOOL; // 0: Kabinentür Einlauf offen ST175
    I9001_ST175_kabinentur_auslauf_offen      AT %I* : BOOL; // 1: Kabinentür Auslauf offen ST175
    I9002_ST180_entlad_fullstandskontroll_box AT %I* : BOOL; // 2: Entlade-& Füllstandskontrolle Box ST180

    //-5017
    (* pnp ST180 *)
    I9100_ST180_greifer_patrone_links_zu         AT %I* : BOOL; // 0: ST180 Greifer Patrone links zu
    I9101_ST180_greifer_patrone_links_offen      AT %I* : BOOL; // 1: ST180 Greifer Patrone links offen
    I9102_ST180_greifer_patrone_rechts_zu        AT %I* : BOOL; // 2: ST180 Greifer Patrone rechts zu
    I9103_ST180_greifer_patrone_rechts_offen     AT %I* : BOOL; // 3: ST180 Greifer Patrone rechts offen
    I9104_ST180_niederhalter_deckel_links_oben   AT %I* : BOOL; // 4: ST180 Niederhalter Deckel links oben
    I9105_ST180_niederhalter_deckel_links_unten  AT %I* : BOOL; // 5: ST180 Niederhalter Deckel links unten
    I9106_ST180_niederhalter_deckel_rechts_oben  AT %I* : BOOL; // 6: ST180 Niederhalter Deckel rechts oben
    I9107_ST180_niederhalter_deckel_rechts_unten AT %I* : BOOL; // 7: ST180 Niederhalter Deckel rechts unten

    //-5018
    (* pnp ST185 *)
    I9200_ST185_greifer_patrone_links_zu         AT %I* : BOOL; // 0: ST185 Greifer Patrone links zu
    I9201_ST185_greifer_patrone_links_offen      AT %I* : BOOL; // 1: ST185 Greifer Patrone links offen
    I9202_ST185_greifer_patrone_rechts_zu        AT %I* : BOOL; // 2: ST185 Greifer Patrone rechts zu
    I9203_ST185_greifer_patrone_rechts_offen     AT %I* : BOOL; // 3: ST185 Greifer Patrone rechts offen
    I9204_ST185_niederhalter_deckel_links_oben   AT %I* : BOOL; // 4: ST185 Niederhalter Deckel links oben
    I9205_ST185_niederhalter_deckel_links_unten  AT %I* : BOOL; // 5: ST185 Niederhalter Deckel links unten
    I9206_ST185_niederhalter_deckel_rechts_oben  AT %I* : BOOL; // 6: ST185 Niederhalter Deckel rechts oben
    I9207_ST185_niederhalter_deckel_rechts_unten AT %I* : BOOL; // 7: ST185 Niederhalter Deckel rechts unten

    //-10960B2
    (* Wegmesssenor ST175 *)
    I9300_ST175_wegmesssensor AT %I* : UINT; // 0: Wegmesssenor ST175

    //-15506
    (* feeder ST105 *)
    Q9500_ST105_Freigabe_WF         AT %Q* : BOOL; // 1: Run vibrator feeder (nearest of the rotary table)
    Q9501_ST105_Freigabe_LF         AT %Q* : BOOL; // 2 Run LF 
    I9502_ST105_Fullstand_kontrolle AT %I* : BOOL; // 3: vibrator full of piece sensor

END_VAR

// ---- GVLs/OUT.TcGVL
{attribute 'qualified_only'}
VAR_GLOBAL
    (*******************************************************************)
    (* AUSGÄNGE *)
    (*******************************************************************)
    (* Modul *)

    // 170D2
    Q000_ AT %QX0.0 : BOOL; // 
    Q001_ AT %QX0.1 : BOOL; // 
    Q002_ AT %QX0.2 : BOOL; // 
    Q003_ AT %QX0.3 : BOOL; // 
    Q004_ AT %QX0.4 : BOOL; // 
    Q005_ AT %QX0.5 : BOOL; // 
    Q006_ AT %QX0.6 : BOOL; // 
    Q007_ AT %QX0.7 : BOOL; // 

    Q010_     AT %QX1.0  : BOOL; // Sauger LN 230 Start
    Q011_                        AT %QX1.1  : BOOL; // 
    Q012_                             AT %QX1.2 : BOOL; // 
    Q013_                        AT %QX1.3  : BOOL; // 
    Q014_                             AT %QX1.4 : BOOL; // 
    Q015_                        AT %QX1.5  : BOOL; // 
    Q016_                             AT %QX1.6 : BOOL; // 
    Q017_                        AT %QX1.7  : BOOL; // 

    // 170D7
    Q020_ST150_ultraschall_start AT %QX02.0 : BOOL; // Ultraschall 150.20 Start
    Q021_ST150_ultraschall_reset AT %QX02.1 : BOOL; // Ultraschall 150.20 Reset
    Q022_ST150_ultraschall_data_bit_0
        AT %QX02.2                               : BOOL; // Ultraschall 150.20 Data HEX1
    Q023_ST150_ultraschall_data_bit_1 AT %QX02.3 : BOOL; // Ultraschall 150.20 Data HEX2
    Q024_ST150_ultraschall_data_bit_2 AT %QX02.4 : BOOL; // Ultraschall 150.20 Data HEX4
    Q025_ST150_ultraschall_data_bit_3 AT %QX02.5 : BOOL; // Ultraschall 150.20 Data HEX8
    Q026_ST170_rfid_start_links       AT %QX02.6 : BOOL; // RFID Test links 170.20
    Q027_ST170_rfid_start_rechts      AT %QX02.7 : BOOL; // RFID Test rechts 170.21

    Q030_ST155_ultraschall_start      AT %QX03.0 : BOOL; // Ultraschall 155.20 Start    
    Q031_ST155_ultraschall_reset      AT %QX03.1 : BOOL; // Ultraschall 155.20 Reset    
    Q032_ST155_ultraschall_data_bit_0 AT %QX03.2 : BOOL; // Ultraschall 155.20 Data HEX1
    Q033_ST155_ultraschall_data_bit_1 AT %QX03.3 : BOOL; // Ultraschall 155.20 Data HEX2
    Q034_ST155_ultraschall_data_bit_2 AT %QX03.4 : BOOL; // Ultraschall 155.20 Data HEX4
    Q035_ST155_ultraschall_data_bit_3 AT %QX03.5 : BOOL; // Ultraschall 155.20 Data HEX8
    Q036_                             AT %QX03.6 : BOOL; // 
    Q037_                             AT %QX03.7 : BOOL; // 

    // 171D2
    Q040_ST170_RFID_Links_Type_Bit_0  AT %QX04.0 : BOOL; // Bit 0 of the RFID type
    Q041_ST170_RFID_Links_Type_Bit_1  AT %QX04.1 : BOOL; // Bit 1 of the RFID type
    Q042_ST170_RFID_Links_Type_Bit_2  AT %QX04.2 : BOOL; // Bit 2 of the RFID type
    Q043_ST170_RFID_Rechts_Type_Bit_0 AT %QX04.3 : BOOL; // Bit 0 of the RFID type
    Q044_ST170_RFID_Rechts_Type_Bit_1 AT %QX04.4 : BOOL; // Bit 1 of the RFID type
    Q045_ST170_RFID_Rechts_Type_Bit_2 AT %QX04.5 : BOOL; // Bit 2 of the RFID type
    Q046_                             AT %QX04.6 : BOOL; // 
    Q047_                      AT %QX04.7 : BOOL; // 

    Q050_ AT %QX05.0 : BOOL; // 
    Q051_ AT %QX05.1 : BOOL; // 
    Q052_ AT %QX05.2 : BOOL; // 
    Q053_ AT %QX05.3 : BOOL; // 
    Q054_ AT %QX05.4 : BOOL; // 
    Q055_ AT %QX05.5 : BOOL; // 
    Q056_ AT %QX05.6 : BOOL; // 
    Q057_ AT %QX05.7 : BOOL; // 

    // 10170D2
    Q100_ST175_laser_fernschalfung AT %QX10.0 : BOOL; // Laser Fernschalfung
    Q101_ST175_Sauger_LN_230_Start         AT %QX10.1 : BOOL; // Sauger Laser 175.21 Start
    Q102_ST185_entladen_ein        AT %QX10.2 : BOOL; // Entladeband 185.21 ein
    Q103_Doppel_tur_lock           AT %QX10.3 : BOOL; // Doppel Türe 5+6 Verriegelung
    Q104_ST110_vacum_on_left       AT %QX10.4 : BOOL; // ST110 Vacum greifer left on 
    Q105_ST110_vacum_on_right      AT %QX10.5 : BOOL; // ST110 Vacum greifer right on 
    Q107_                          AT %QX10.7 : BOOL; // Reserve
    Q106_ST105_zusatz_band_on      AT %QX10.6 : BOOL; // ST105 band between bowl and linear feeder

    Q110_ AT %QX11.0 : BOOL; // Reserve
    Q111_ AT %QX11.1 : BOOL; // Reserve
    Q112_ AT %QX11.2 : BOOL; // Reserve
    Q113_ AT %QX11.3 : BOOL; // Reserve
    Q114_ AT %QX11.4 : BOOL; // Reserve
    Q115_ AT %QX11.5 : BOOL; // Reserve
    Q116_ AT %QX11.6 : BOOL; // Reserve
    Q117_ AT %QX11.7 : BOOL; // Reserve

    // 10170D7
    Q120_ AT %QX12.0 : BOOL; // 
    Q121_ AT %QX12.1 : BOOL; // 
    Q122_ AT %QX12.2 : BOOL; // 
    Q123_ AT %QX12.3 : BOOL; // 
    Q124_ AT %QX12.4 : BOOL; // 
    Q125_ AT %QX12.5 : BOOL; // 
    Q126_ AT %QX12.6 : BOOL; // 
    Q127_ AT %QX12.7 : BOOL; // 

    Q130_ AT %QX13.0 : BOOL; // 
    Q131_ AT %QX13.1 : BOOL; // 
    Q132_ AT %QX13.2 : BOOL; // 
    Q133_ AT %QX13.3 : BOOL; // 
    Q134_ AT %QX13.4 : BOOL; // 
    Q135_ AT %QX13.5 : BOOL; // 
    Q136_ AT %QX13.6 : BOOL; // 
    Q137_ AT %QX13.7 : BOOL; // 

    // analog
    QA01_ST130_pressure_valve_left  AT %Q* : UINT; // Pro.Druckregelventil left
    QA02_ST130_pressure_valve_right AT %Q* : UINT; // Pro.Druckregelventil right
    QA03_ST135_pressure_valve_left  AT %Q* : UINT; // Pro.Druckregelventil left
    QA04_ST135_pressure_valve_right AT %Q* : UINT; // Pro.Druckregelventil right

    Q_CPX9_1_EnergiEin_led   AT %Q* : BOOL; // Blue button on the panel
    Q_CPX9_1_Process_running AT %Q* : BOOL; // Green button on the panel
    Q_CPX9_1_Process_stopped AT %Q* : BOOL; // Red button on the panel

END_VAR

// ---- GVLs/PERS.TcGVL
{attribute 'qualified_only'}
VAR_GLOBAL RETAIN PERSISTENT
    (***********************************************************************************************)
    (* COUNTER *)
    (***********************************************************************************************)
    //COUNTER 
    udiTotalOK  : UDINT; // Total Counter  OK 
    udiTotalNOK : UDINT; // Total Counter  NOK 

    udiTempOK  : UDINT; // Temporary Counter  OK 
    udiTempNOK : UDINT; // Temporary Counter  NOK 

    //OPERATING HOURS
    udiCountHon    : UDINT; // Operating hours SYSTEM POWER ON [h] 
    udiCount6Mon   : UDINT; // Operating hours SYSTEM POWER ON [6min (0.1h)] 
    udiCountHauto  : UDINT; // Operating hours SYSTEM IN AUTOMATIC MODE [h] 
    udiCount6Mauto : UDINT; // Operating hours SYSTEM IN AUTOMATIC MODE [6min (0.1h)] 

    (***********************************************************************************************)
    (* PARAMETER *)
    (***********************************************************************************************)
    udiArCntST00 : ARRAY[0..4] OF UDINT; (* Counter ST00 
															0:
	*)
    (***********************************************************************************************)
    (* Timer *)
    (***********************************************************************************************)
    //Zylinder																		
    dwArTimeZylST01 : ARRAY[0..20] OF DWORD; (* Time Zylinder Station 01
																0: GENERAL
																1: 
	*)
    //Diverse
    dwArTimeST00 : ARRAY[0..10] OF DWORD; (* Time zur ST00
                                                            0:
                                                            1:  
                                                        *)

    (***********************************************************************************************)
    (* Werte *)
    (***********************************************************************************************)
    iWTstat : ARRAY[1..10] OF INT; (* STATUS WT [Station]
																<0: NIO
																 0: LEER
																>0: STATION
															*)

    (***********************************************************************************************)
    (* Application *)
    (***********************************************************************************************)

    {attribute 'to_json'}
    iStationTimeDef1 : ARRAY[1..CONST.STATION_NUMBER] OF DINT;
    {attribute 'to_json'}
    iStationTimeDef2 : ARRAY[1..CONST.STATION_NUMBER] OF DINT;

    //{attribute 'to_json'}
    //_20_AUTO.recipe : Recipe_21_101_t;

    {attribute 'to_json'}
    recipeList : ARRAY[0..CONST.MAX_RECIPE_NUMBER] OF Recipe_21_101_t; // registery of recipe
	
    eRecipeCurrent : RecipeType_e; // selected recipe to be executed
	
    {attribute 'to_json'}
    iRecipeCurrent : INT; // selected recipe to be executed

END_VAR

// ---- GVLs/SIMU.TcGVL
{attribute 'qualified_only'}
VAR_GLOBAL
    iCompletionHMI : ARRAY[0..CONST.STATION_NUMBER] OF INT;

    lrSpeedMover       : LREAL := 20.0;
    lrAccelMover       : LREAL; // is lrAccelMoverSlider^2
    lrAccelMoverSlider : LREAL := 0.4;
	
	axis_ref : ARRAY [0..Axis_e._max-1] OF AXIS_REF;
	
	sLaserFileName : STRING;
	iLaserFileNum : INT := 1000;
END_VAR

// ---- POUs/20_AUTO/BuR SuperTrack com/gMoverAxis.TcGVL
{attribute 'qualified_only'}
VAR_GLOBAL
    I_BuR_MoverAxis    AT %I* : BuR_MoverAxis_Array_u; // all the movers
    Q_CT_Shuttle_to_BR AT %Q* : CT_Shuttle_Tc_to_BR_u;
    I_CT_Track_from_BR AT %I* : CT_Track_BR_to_Tc_u;
    Q_CT_Track_to_BR   AT %Q* : CT_Track_Tc_to_BR_u;

END_VAR

// ---- POUs/20_AUTO/ST105/ST105_Axis.TcGVL
{attribute 'qualified_only'}
VAR_GLOBAL CONSTANT
    const105_11Z : AxisLinMotConst_t := (POS_MIN := 0, POS_MAX := 200, VELO_MAX := 1500, VELO_MANU := 50);
    const105_10W : AxisLinMotConst_t := (POS_MIN := 0, POS_MAX := 360, VELO_MAX := 720, VELO_MANU := 50);

END_VAR
VAR_GLOBAL
    axis105_11Z : AxisLinMot_t;
    axis105_10W : AxisLinMot_t;
END_VAR
VAR_GLOBAL RETAIN
    // Recipe values are managed elsewhere
END_VAR

// ---- POUs/20_AUTO/ST110/ST110_Axis.TcGVL
{attribute 'qualified_only'}
VAR_GLOBAL CONSTANT
    const110_01Y : AxisLinMotConst_t := (POS_MIN := 0, POS_MAX := 220, VELO_MAX := 1500, VELO_MANU := 100);
    const110_02Z : AxisLinMotConst_t := (POS_MIN := 0, POS_MAX := 200, VELO_MAX := 1500, VELO_MANU := 50);
    const110_03Z : AxisLinMotConst_t := (POS_MIN := 0, POS_MAX := 200, VELO_MAX := 1500, VELO_MANU := 50);
    const110_04Z : AxisLinMotConst_t := (POS_MIN := 0, POS_MAX := 200, VELO_MAX := 1500, VELO_MANU := 50);
    const110_10W : AxisLinMotConst_t := (POS_MIN := 0, POS_MAX := 360, VELO_MAX := 720, VELO_MANU := 50);

END_VAR
VAR_GLOBAL
    axis110_01Y : AxisLinMot_t;
    axis110_02Z : AxisBeckhoff_t;
    axis110_03Z : AxisBeckhoff_t;
    axis110_04Z : AxisBeckhoff_t;
    axis110_10W : AxisLinMot_t;
END_VAR
VAR_GLOBAL RETAIN
    // Recipe values are managed elsewhere
END_VAR

// ---- POUs/20_AUTO/ST115/ST115_Axis.TcGVL
{attribute 'qualified_only'}
VAR_GLOBAL CONSTANT
    const115_01Y : AxisLinMotConst_t := (POS_MIN := -5, POS_MAX := 650, VELO_MAX := 2000, VELO_MANU := 100);
    const115_02Z : AxisLinMotConst_t := (POS_MIN := -5, POS_MAX := 650, VELO_MAX := 2000, VELO_MANU := 50);
    const115_03Z : AxisLinMotConst_t := (POS_MIN := -5, POS_MAX := 650, VELO_MAX := 2000, VELO_MANU := 50);
    const115_10W : AxisLinMotConst_t := (POS_MIN := 0, POS_MAX := 360, VELO_MAX := 360, VELO_MANU := 50);

END_VAR
VAR_GLOBAL
    axis115_01Y : AxisLinMot_t;
    axis115_02Z : AxisBeckhoff_t;
    axis115_03Z : AxisBeckhoff_t;
    axis115_04Z : AxisBeckhoff_t;
    axis115_10W : AxisLinMot_t;
END_VAR
VAR_GLOBAL RETAIN
    // Recipe values are managed elsewhere
END_VAR

// ---- POUs/20_AUTO/ST120/ST120_Axis.TcGVL
{attribute 'qualified_only'}
VAR_GLOBAL CONSTANT
    const120_01Y : AxisLinMotConst_t := (POS_MIN := -5, POS_MAX := 450, VELO_MAX := 2000, VELO_MANU := 100);
    const120_02Z : AxisLinMotConst_t := (POS_MIN := -5, POS_MAX := 650, VELO_MAX := 2000, VELO_MANU := 50);

END_VAR
VAR_GLOBAL
    axis120_01Y : AxisLinMot_t;
    axis120_02Z : AxisLinMot_t;
END_VAR
VAR_GLOBAL RETAIN
    // Recipe values are managed elsewhere
END_VAR

// ---- POUs/20_AUTO/ST125/ST125_Axis.TcGVL
{attribute 'qualified_only'}
VAR_GLOBAL CONSTANT
    const125_01Y : AxisLinMotConst_t := (POS_MIN := -5, POS_MAX := 200, VELO_MAX := 2000, VELO_MANU := 100);
    const125_02Z : AxisLinMotConst_t := (POS_MIN := -5, POS_MAX := 200, VELO_MAX := 2000, VELO_MANU := 50);
    const125_10W : AxisLinMotConst_t := (POS_MIN := 0, POS_MAX := 360, VELO_MAX := 720, VELO_MANU := 50);

END_VAR
VAR_GLOBAL
    axis125_01Y : AxisLinMot_t;
    axis125_02Z : AxisLinMot_t;
    axis125_10W : AxisLinMot_t;
END_VAR
VAR_GLOBAL RETAIN
    // Recipe values are managed elsewhere
END_VAR

// ---- POUs/20_AUTO/ST130/ST130_Axis.TcGVL
{attribute 'qualified_only'}
VAR_GLOBAL CONSTANT
    const130_01Z : AxisLinMotConst_t := (POS_MIN := -5, POS_MAX := 200, VELO_MAX := 2000, VELO_MANU := 50);
    const130_10Z : AxisLinMotConst_t := (POS_MIN := -5, POS_MAX := 150, VELO_MAX := 2000, VELO_MANU := 50);

END_VAR
VAR_GLOBAL
    axis130_01Z : AxisBeckhoff_t;
    axis130_10Z : AxisLinMot_t;
END_VAR
VAR_GLOBAL RETAIN
    // Recipe values are managed elsewhere
END_VAR

// ---- POUs/20_AUTO/ST145/ST145_Axis.TcGVL
{attribute 'qualified_only'}
VAR_GLOBAL CONSTANT
    const145_01Y : AxisLinMotConst_t := (POS_MIN := -5, POS_MAX := 200, VELO_MAX := 2000, VELO_MANU := 50);
    const145_02Z : AxisLinMotConst_t := (POS_MIN := -5, POS_MAX := 150, VELO_MAX := 2000, VELO_MANU := 50);
    const145_10W : AxisLinMotConst_t := (POS_MIN := 0, POS_MAX := 360, VELO_MAX := 360, VELO_MANU := 50);

END_VAR
VAR_GLOBAL
    axis145_01Y : AxisLinMot_t;
    axis145_02Z : AxisLinMot_t;
    axis145_10W : AxisLinMot_t;
END_VAR
VAR_GLOBAL RETAIN
    // Recipe values are managed elsewhere
END_VAR

// ---- POUs/20_AUTO/ST16x/CETA/CETA_IO.TcGVL
{attribute 'qualified_only'}
VAR_GLOBAL
    I_ST160_StatusBits  AT %I* : CETA_IN_u;            // connect this to the 2 first byte of the input of the CETATEST
    I_ST160_Data        AT %I* : ARRAY[0..61] OF BYTE; // connect those 62 bytes right after xIN_StatusBits
    Q_ST160_CommandBits AT %Q* : CETA_OUT_u;           // connect this to the 2 first byte of the Output of the CETATEST
    Q_ST160_Data        AT %Q* : ARRAY[0..29] OF BYTE; // connect those 30 bytes right after xIN_StatusBits
	
    I_ST165_StatusBits  AT %I* : CETA_IN_u;            // connect this to the 2 first byte of the input of the CETATEST
    I_ST165_Data        AT %I* : ARRAY[0..61] OF BYTE; // connect those 62 bytes right after xIN_StatusBits
    Q_ST165_CommandBits AT %Q* : CETA_OUT_u;           // connect this to the 2 first byte of the Output of the CETATEST
    Q_ST165_Data        AT %Q* : ARRAY[0..29] OF BYTE; // connect those 30 bytes right after xIN_StatusBits
END_VAR

// ---- POUs/20_AUTO/ST16x/ST16x_Axis.TcGVL
{attribute 'qualified_only'}
VAR_GLOBAL CONSTANT
    const160_01Z : AxisLinMotConst_t := (POS_MIN := 0, POS_MAX := 220, VELO_MAX := 1500, VELO_MANU := 50);
    const165_01Z : AxisLinMotConst_t := (POS_MIN := 0, POS_MAX := 220, VELO_MAX := 1500, VELO_MANU := 50);
END_VAR
VAR_GLOBAL
    axis160_01Z : AxisBeckhoff_t;
    axis165_01Z : AxisBeckhoff_t;
END_VAR
VAR_GLOBAL RETAIN
    // Recipe values are managed elsewhere
END_VAR

// ---- POUs/20_AUTO/ST175/Trumpf/if_TruMark.TcGVL
{attribute 'qualified_only' := ''}
VAR_GLOBAL
	// starts a TLV command
	bTlvCmd: BOOL;
	// starts a BIT command
	bBitCmd: BOOL;
	// reset error
	bResetErr: BOOL;
	// input parameter for TLV command
	diTlvTag: DINT;
	// input parameter for TLV command
	sTlvValueIn: STRING;
	// input parameter for BIT command	(32 bit)
	dwBitIn: DWORD;
	// indicates if TruMark_Profibus is running
	bBusy: BOOL;
	// indicates if an error (Communication / Bussystem) is occured
	bError: BOOL;
	sErrorMsg: STRING;
	// return code of a TLV command
	byTlvReturnCode: BYTE;
	// return value of a TLV command
	sTlvRespons: STRING;
	// extended error code
	byTlvExtErrCode: BYTE;
	// current status
	Status: TruMarkLaserStatus;
END_VAR

// ---- POUs/20_AUTO/ST180/ST180_Axis.TcGVL
{attribute 'qualified_only'}
VAR_GLOBAL CONSTANT
    const180_01Y : AxisLinMotConst_t := (POS_MIN := -5, POS_MAX := 250, VELO_MAX := 2000, VELO_MANU := 100);
    const180_02Z : AxisLinMotConst_t := (POS_MIN := -5, POS_MAX := 320, VELO_MAX := 2000, VELO_MANU := 50);
    const180_10Z : AxisLinMotConst_t := (POS_MIN := -5, POS_MAX := 200, VELO_MAX := 2000, VELO_MANU := 50);

END_VAR
VAR_GLOBAL
    axis180_01Y : AxisLinMot_t;
    axis180_02Z : AxisLinMot_t;
    axis180_10Z : AxisLinMot_t;
END_VAR
VAR_GLOBAL RETAIN
    // Recipe values are managed elsewhere
END_VAR

// ---- POUs/20_AUTO/ST185/ST185_Axis.TcGVL
{attribute 'qualified_only'}
VAR_GLOBAL CONSTANT
    const185_01Y : AxisLinMotConst_t := (POS_MIN := -5, POS_MAX := 250, VELO_MAX := 2000, VELO_MANU := 100);
    const185_02Z : AxisLinMotConst_t := (POS_MIN := -5, POS_MAX := 300, VELO_MAX := 2000, VELO_MANU := 50);
    const185_10Z : AxisLinMotConst_t := (POS_MIN := -5, POS_MAX := 200, VELO_MAX := 2000, VELO_MANU := 50);

END_VAR
VAR_GLOBAL
    axis185_01Y : AxisLinMot_t;
    axis185_02Z : AxisLinMot_t;
    axis185_10Z : AxisLinMot_t;
END_VAR
VAR_GLOBAL RETAIN
    // Recipe values are managed elsewhere
END_VAR

// ---- POUs/20_AUTO/Mover/ISimuMoverTimers.TcIO
INTERFACE ISimuMoverTimers

(* Process time, expressed in milisecond *)
PROPERTY iProcessTimeMili_1 : DINT
GET
END_GET
SET
END_SET
END_PROPERTY

(* Process time, expressed in milisecond *)
PROPERTY iProcessTimeMili_2 : DINT
GET
END_GET
SET
END_SET
END_PROPERTY

END_INTERFACE

// ---- POUs/20_AUTO/Mover/IStation.TcIO
INTERFACE IStation

PROPERTY Position : REFERENCE TO FB_Position
GET
END_GET
SET
END_SET
END_PROPERTY

PROPERTY Process : REFERENCE TO FB_AUT_ABSTRACT
GET
END_GET
SET
END_SET
END_PROPERTY

END_INTERFACE

// ---- POUs/20_AUTO/TOOL/IObject.TcIO
// Basic object interface that provide core function for each FB
INTERFACE IObject

METHOD Equals : BOOL
VAR_INPUT
	object : REFERENCE TO IObject;
END_VAR
END_METHOD

METHOD ToString : STRING
VAR_INPUT
END_VAR
END_METHOD

END_INTERFACE

// ---- POUs/00_MAIN/MAIN.TcPOU
PROGRAM MAIN
VAR
	MoverMan	: FB_MoverMan;
END_VAR

_02_SAFETY();
_05_FLAGS( xIN_AIR:=TRUE, xIN_btRES_TEMP:=HMI.btArMain[8]);

//HMI
_10_HMI();

MoverMan();

//AUTO
_20_AUTO(xIN_Quit:= _14_STATE._FB_btQUIT.pbtIN^.rtrig , enIN_State:= HMI.enState);

END_PROGRAM

// ---- POUs/20_AUTO/Mover/FB_MoverMan.TcPOU
FUNCTION_BLOCK FB_MoverMan
VAR_INPUT
END_VAR
VAR_OUTPUT
    xOUT_AllMoverEmpty : BOOL; // TRUE when LastStationVisited from all shuttle are 0
    xOUT_Error         : BOOL; // CleverTrack is in error and needs a reset
END_VAR
VAR
    _PieceHolderList : ARRAY[1..2] OF FB_PieceHolder[(0),
                                                     (0)];
    _SimuMoverList : ARRAY[1..19] OF FB_SimuMoverAxis[(116),
                                                      (433),
                                                      (750),
                                                      (1067),
                                                      (1384),
                                                      (1701),
                                                      (2018),
                                                      (2335),
                                                      (2652),
                                                      (3000),
                                                      (3400),
                                                      (3800),
                                                      (5200),
                                                      (5600),
                                                      (6000),
                                                      (6400),
                                                      (6800),
                                                      (7200),
                                                      (7600)];

    _MoverList : ARRAY[1..19] OF FB_Mover[(1, _SimuMoverList[1]),
                                          (2, _SimuMoverList[2]),
                                          (3, _SimuMoverList[3]),
                                          (4, _SimuMoverList[4]),
                                          (5, _SimuMoverList[5]),
                                          (6, _SimuMoverList[6]),
                                          (7, _SimuMoverList[7]),
                                          (8, _SimuMoverList[8]),
                                          (9, _SimuMoverList[9]),
                                          (10, _SimuMoverList[10]),
                                          (11, _SimuMoverList[11]),
                                          (12, _SimuMoverList[12]),
                                          (13, _SimuMoverList[13]),
                                          (14, _SimuMoverList[14]),
                                          (15, _SimuMoverList[15]),
                                          (16, _SimuMoverList[16]),
                                          (17, _SimuMoverList[17]),
                                          (18, _SimuMoverList[18]),
                                          (19, _SimuMoverList[19])];

    _PosList : ARRAY[1..CONST.STATION_NUMBER] OF FB_Position[(125, 1, 1),
                                                             (625, 1, 1),
                                                             (1125, 1, 1),
                                                             (1375, 1, 1),
                                                             (1625, 1, 1),
                                                             (1875, 1, 1),
                                                             (2375, 1, 1),
                                                             (2625, 1, 1),
                                                             (2875, 1, 1),
                                                             (3125, 1, 1),
                                                             (3625, 1, 1),
                                                             (3875, 1, 1),
                                                             // second part
                                                             (5205, 1, 1),
                                                             (5455, 1, 1),
                                                             (6165, 1, 1),
                                                             (6830, 1, 1), // waiting pos
                                                             (7365, 1, 1),
                                                             (7695, 1, 1),
                                                             (8655, 1, 1),
                                                             (8905, 1, 1)];

    _StationList : ARRAY[1..CONST.STATION_NUMBER] OF
        FB_Station[(_PosList[1],
                    GVL.st105_aut,
                    -250,
                    ApproachScenario_e.WaitOnFinishedProcess,
                    3,
                    5),
                   (_PosList[2],
                    GVL.st110_aut,
                    -250,
                    ApproachScenario_e.WaitOnFinishedProcess,
                    1,
                    10),
                   (_PosList[3],
                    GVL.st115_aut,
                    -250,
                    ApproachScenario_e.WaitOnFinishedProcess,
                    1,
                    15),
                   (_PosList[4],
                    GVL.st120_aut,
                    0,
                    ApproachScenario_e.WaitOnFinishedProcess,
                    0,
                    20),
                   (_PosList[5],
                    GVL.st125_aut,
                    0,
                    ApproachScenario_e.WaitOnFinishedProcess,
                    3,
                    25),
                   (_PosList[6],
                    GVL.st128_aut,
                    -100,
                    ApproachScenario_e.WaitOnFinishedProcess,
                    1,
                    28),
                   (_PosList[7],
                    GVL.st130_aut,
                    0,
                    ApproachScenario_e.WaitOnFinishedProcess,
                    1,
                    30),
                   (_PosList[8],
                    GVL.st135_aut,
                    0,
                    ApproachScenario_e.WaitOnFinishedProcess,
                    3,
                    35),
                   (_PosList[9],
                    GVL.st140_aut,
                    -100,
                    ApproachScenario_e.DoNotWait,
                    0,
                    40),
                   (_PosList[10],
                    GVL.st145_aut,
                    0,
                    ApproachScenario_e.WaitOnFinishedProcess,
                    0,
                    45),
                   (_PosList[11],
                    GVL.st150_aut,
                    -250,
                    ApproachScenario_e.WaitOnFinishedProcess,
                    1,
                    50),
                   (_PosList[12],
                    GVL.st155_aut,
                    -500,
                    ApproachScenario_e.WaitOnFinishedProcess,
                    1,
                    55),
                   (_PosList[13],
                    GVL.st160_aut,
                    -250,
                    ApproachScenario_e.WaitOnFinishedProcess,
                    3,
                    60),
                   (_PosList[14],
                    GVL.st165_aut,
                    -500,
                    ApproachScenario_e.WaitOnFinishedProcess,
                    3,
                    65),
                   (_PosList[15],
                    GVL.st170_aut,
                    -250,
                    ApproachScenario_e.WaitOnFinishedProcess,
                    2,
                    70),
                   (_PosList[16],
                    0,
                    0,
                    ApproachScenario_e.DoNotWait,
                    3,
                    74),
                   (_PosList[17],
                    GVL.st175_aut,
                    0,
                    ApproachScenario_e.WaitOnFreeStation,
                    0,
                    75),
                   (_PosList[18],
                    GVL.st176_aut,
                    0,
                    ApproachScenario_e.WaitOnFinishedProcess,
                    0,
                    76),
                   (_PosList[19],
                    GVL.st180_aut,
                    -400,
                    ApproachScenario_e.WaitOnFinishedProcess,
                    2,
                    80),
                   (_PosList[20],
                    GVL.st185_aut,
                    0,
                    ApproachScenario_e.WaitOnFinishedProcess,
                    3,
                    85)];

    // Smart
    _StationSet1 :
        ARRAY[1..CONST.STATION_NUMBER] OF INT := [0,  // ST105
                                                  0,  // ST110
                                                  -1, // ST115
                                                  -1, // ST120
                                                  0,  // ST125
                                                  0,  // ST128
                                                  1,  // ST130
                                                  -1, // ST135
                                                  0,  // ST140
                                                  0,  // ST145
                                                  2,  // ST150
                                                  0,  // ST155
                                                  3,  // ST160
                                                  3,  // ST165
                                                  0,  // ST170
                                                  0,  // ST174
                                                  4,  // ST175
                                                  -1, // ST176
                                                  0,  // ST180
                                                  0]; // ST185

    // Pro
    _StationSet2 :
        ARRAY[1..CONST.STATION_NUMBER] OF INT := [0,  // ST105
                                                  0,  // ST110
                                                  -1, // ST115
                                                  0,  // ST120
                                                  0,  // ST125
                                                  0,  // ST128
                                                  1,  // ST130
                                                  -1, // ST135
                                                  0,  // ST140
                                                  0,  // ST145
                                                  2,  // ST150
                                                  -1, // ST155
                                                  3,  // ST160
                                                  3,  // ST165
                                                  0,  // ST170
                                                  0,  // ST174
                                                  4,  // ST175
                                                  -1, // ST176
                                                  0,  // ST180
                                                  0]; // ST185

    // Mini
    _StationSet3 :
        ARRAY[1..CONST.STATION_NUMBER] OF INT := [0,  // ST105
                                                  0,  // ST110
                                                  -1, // ST115
                                                  -1, // ST120
                                                  0,  // ST125
                                                  0,  // ST128
                                                  1,  // ST130
                                                  -1, // ST135
                                                  0,  // ST140
                                                  0,  // ST145
                                                  2,  // ST150
                                                  0,  // ST155
                                                  3,  // ST160
                                                  3,  // ST165
                                                  0,  // ST170
                                                  0,  // ST174
                                                  4,  // ST175
                                                  -1, // ST176
                                                  0,  // ST180
                                                  0]; // ST185
    // Blue    
    _StationSet4 :
        ARRAY[1..CONST.STATION_NUMBER] OF INT := [0,  // ST105
                                                  -1, // ST110
                                                  -1, // ST115
                                                  -1, // ST120
                                                  0,  // ST125
                                                  0,  // ST128
                                                  1,  // ST130
                                                  -1, // ST135
                                                  0,  // ST140
                                                  0,  // ST145
                                                  2,  // ST150
                                                  0,  // ST155
                                                  3,  // ST160
                                                  3,  // ST165
                                                  -1, // ST170
                                                  0,  // ST174
                                                  4,  // ST175
                                                  -1, // ST176
                                                  0,  // ST180
                                                  0]; // ST185
    _StationSet5 :
        ARRAY[1..CONST.STATION_NUMBER] OF INT := [0,
                                                  0,
                                                  0,
                                                  0,
                                                  0,
                                                  0,
                                                  0,
                                                  0,
                                                  0,
                                                  0,
                                                  0,
                                                  0,
                                                  0,
                                                  0,
                                                  0,
                                                  0,
                                                  0,
                                                  0,
                                                  0,
                                                  0];
    _StationSet6 :
        ARRAY[1..CONST.STATION_NUMBER] OF INT := [0,
                                                  0,
                                                  0,
                                                  0,
                                                  0,
                                                  0,
                                                  0,
                                                  0,
                                                  0,
                                                  0,
                                                  0,
                                                  0,
                                                  0,
                                                  0,
                                                  0,
                                                  0,
                                                  0,
                                                  0,
                                                  0,
                                                  0];
		// Pro Blue
    _StationSet7 :
        ARRAY[1..CONST.STATION_NUMBER] OF INT := [0,  // ST105
                                                  -1, // ST110
                                                  -1, // ST115
                                                  0,  // ST120
                                                  0,  // ST125
                                                  0,  // ST128
                                                  1,  // ST130
                                                  -1, // ST135
                                                  0,  // ST140
                                                  0,  // ST145
                                                  2,  // ST150
                                                  -1, // ST155
                                                  3,  // ST160
                                                  3,  // ST165
                                                  -1, // ST170
                                                  0,  // ST174
                                                  4,  // ST175
                                                  -1, // ST176
                                                  0,  // ST180
                                                  0]; // ST185

    _SelWorkStationList : ARRAY[1..7] OF POINTER TO ARRAY[1..CONST.STATION_NUMBER] OF INT
        := [ADR(_StationSet1), ADR(_StationSet2), ADR(_StationSet3), ADR(_StationSet4), ADR(_StationSet5), ADR(_StationSet6), ADR(_StationSet7)];

    _WorkStationList : ARRAY[1..CONST.MAX_RECIPE_NUMBER] OF
        FB_StationMan[(ADR(_StationList), _SelWorkStationList[1], _PieceHolderList[1]),
                      (ADR(_StationList), _SelWorkStationList[2], _PieceHolderList[1]),
                      (ADR(_StationList), _SelWorkStationList[3], _PieceHolderList[1]),
                      (ADR(_StationList), _SelWorkStationList[4], _PieceHolderList[1]),
                      (ADR(_StationList), _SelWorkStationList[5], _PieceHolderList[1]),
                      (ADR(_StationList), _SelWorkStationList[5], _PieceHolderList[1]),
                      (ADR(_StationList), _SelWorkStationList[7], _PieceHolderList[1]),
                      (ADR(_StationList), _SelWorkStationList[5], _PieceHolderList[1]),
                      (ADR(_StationList), _SelWorkStationList[5], _PieceHolderList[1]),
                      (ADR(_StationList), _SelWorkStationList[5], _PieceHolderList[1]),
                      (ADR(_StationList), _SelWorkStationList[5], _PieceHolderList[1])];

    step : INT := 0; //test step

    PH_num : INT := 1; // piece holder selection

    mv_i                : INT;           // mover index
    bMoverSync          : BOOL := FALSE; // external trigger for movers
    iNumOfMoverOnTheWay : INT;           // temp var to know how many mover there are between a given mover and its next station

    lastEmptyStation : REFERENCE TO FB_Station; // temp var to store the next free station

    HMI_Scenario   : ApproachScenario_e := ApproachScenario_e.WaitOnFinishedProcess;
    HMI_TimeAvg    : DINT               := 1000;
    HMI_TimeMin    : DINT               := 900;
    HMI_TimeMax    : DINT               := 1100;
    HMI_xStopMover : BOOL               := FALSE;
    HMI_iSelMover  : INT                := 1;

    HMI_send_all_shuttle_to_unload : BOOL;

    _iID : INT := 0; // instance ID, is set during FB_Init using the value of _iInstanceCounter 
END_VAR
VAR CONSTANT
    MOVER_NUMBER     : INT  := 18;
    TRACK_SIMULATION : BOOL := FALSE; // Set to true when supertrack is in simulation
END_VAR
VAR_STAT
    _iInstanceCounter : INT := 1; // instance counter
END_VAR

(* ---------------------------------------------------------------------------- *)
(* THIS IS A PARTICULAR IMPLEMENTATION OF CLEVERTRAKLIB. THIS SHOULD BE REMOVED *)
CASE step OF

0: // setup everything
    FOR mv_i := 1 TO MOVER_NUMBER BY 1 DO
        _MoverList[mv_i].SetStation(_WorkStationList[PH_num].GetStartStation(_MoverList[mv_i].MoverAxis.CurrentPos)^);
        _MoverList[mv_i].AttachedPieceHolder REF= _WorkStationList[PH_num].PieceHolder;
    END_FOR

    step := 5;

5: // wait until the whole path is free

    IF gMoverAxis.Q_CT_Track_to_BR.asStruct.bCommand.wholePathFree THEN
        step := 10;
    END_IF
10: // turn power on
    gMoverAxis.Q_CT_Track_to_BR.asStruct.bCommand.enablePower := (HMI.enState <> enState.StateMANU);

    IF gMoverAxis.I_CT_Track_from_BR.asStruct.bStatus.powerOn THEN
        step := 11;
    END_IF

11: // init all mover until they the first shuttle is found
    gMoverAxis.Q_CT_Track_to_BR.asStruct.bCommand.startMoverNumberingSequence := (HMI.enState <> enState.StateMANU);

    IF gMoverAxis.I_CT_Track_from_BR.asStruct.bStatus.allIdSet THEN
        gMoverAxis.Q_CT_Track_to_BR.asStruct.bCommand.setShuttleNumber      := FALSE;
        gMoverAxis.Q_CT_Track_to_BR.asStruct.bCommand.releaseUnknownShuttle := FALSE;
        step                                                                := 13;
    END_IF

    IF gMoverAxis.I_CT_Track_from_BR.asStruct.bStatus.unknownMoverAtTarget1 THEN
        IF IO_BOX.I8604_ST105_first_shuttle_pin OR (TRACK_SIMULATION AND CONST.USE_SIMULATION) THEN
            step := 12;
        ELSE
            gMoverAxis.Q_CT_Track_to_BR.asStruct.bCommand.releaseUnknownShuttle := TRUE;
        END_IF
    ELSE
        gMoverAxis.Q_CT_Track_to_BR.asStruct.bCommand.releaseUnknownShuttle := FALSE;
    END_IF

12: // set all id since the first is found
    IF gMoverAxis.I_CT_Track_from_BR.asStruct.bStatus.unknownMoverAtTarget1 THEN
        gMoverAxis.Q_CT_Track_to_BR.asStruct.bCommand.setShuttleNumber := TRUE;
    ELSE
        gMoverAxis.Q_CT_Track_to_BR.asStruct.bCommand.setShuttleNumber := FALSE;
    END_IF

    IF gMoverAxis.I_CT_Track_from_BR.asStruct.bStatus.allIdSet THEN
        gMoverAxis.Q_CT_Track_to_BR.asStruct.bCommand.setShuttleNumber      := FALSE;
        gMoverAxis.Q_CT_Track_to_BR.asStruct.bCommand.releaseUnknownShuttle := FALSE;
        step                                                                := 13;
    END_IF

13: // stop id attrib sequence
    gMoverAxis.Q_CT_Track_to_BR.asStruct.bCommand.startMoverNumberingSequence := FALSE;
    step                                                                      := 14;

14: // check parameter
    // TODO here we have clearly somthing that will not work
    // when using groups... Groups should use the first station to set the waiting position
    // of the whole group
    IF THIS^.CheckWaitPosNotBehindStation() THEN
        ASSERT(0);
    END_IF

    gMoverAxis.Q_CT_Track_to_BR.asStruct.bCommand.enableProcess := TRUE;
    step                                                        := 15;

15: //move every shuttle to the last station
    FOR mv_i := 1 TO MOVER_NUMBER BY 1 DO
        _MoverList[mv_i].SetStation(THIS^._StationList[CONST.STATION_NUMBER]);
        _MoverList[mv_i].MoveToStation();
    END_FOR

    step := 16;
16:
    IF HMI_send_all_shuttle_to_unload THEN
        step := 15;
    END_IF
// do nothing, init done

END_CASE

(* ---------------------------------------------------------------------------- *)

// should be done elsewhere ...
SIMU.lrAccelMover := SIMU.lrAccelMoverSlider * SIMU.lrAccelMoverSlider;

PH_num := PERS.iRecipeCurrent + 1;

// Affect station offset depending on the station offset list
FOR mv_i := 1 TO CONST.STATION_NUMBER BY 1 DO
    _StationList[mv_i].Offset := PERS.recipeList[PERS.iRecipeCurrent].stationOffsets[mv_i - 1];
END_FOR

FOR mv_i := 1 TO MOVER_NUMBER BY 1 DO
    _MoverList[mv_i].AttachedPieceHolder REF= _WorkStationList[PH_num].PieceHolder;

    IF HMI.enState = enState.StateAUTO OR HMI.enState = enState.StateSTEP OR HMI.enState = enState.StateLEER THEN

        CASE _MoverList[mv_i].State OF

        MoverState_e.OperationDone:
            IF __ISVALIDREF(_MoverList[mv_i].Station.Process) THEN
                _MoverList[mv_i].Station.Process.TakeMover();
            ELSE
                ASSERT(0);
            END_IF

            _MoverList[mv_i].SetStation(_WorkStationList[PH_num].GetNextStation(_MoverList[mv_i].Station));

        MoverState_e.WaitOnNextStation:
            // depending on the next station scenario, move
            CASE _MoverList[mv_i].Station.ApproachScenario OF
            // do not wait
            ApproachScenario_e.DoNotWait:
                _MoverList[mv_i].MoveToStation();

            // wait on the next station to be free
            ApproachScenario_e.WaitOnFinishedProcess:
                // Are we in a waiting spot ?
                IF __ISVALIDREF(_MoverList[mv_i].Station.Process) THEN

                    iNumOfMoverOnTheWay := THIS^.GetNumOfMoverOnTheWay(_MoverList[mv_i]);

                    IF 0 = iNumOfMoverOnTheWay THEN
                        _MoverList[mv_i].MoveToStation();

                    ELSIF iNumOfMoverOnTheWay <= _MoverList[mv_i].Station.iMaxWaitingMovers THEN
                        _MoverList[mv_i].MoveToWaitSpot();
                    END_IF

                ELSE
                    _MoverList[mv_i]
                        .SetStation(_WorkStationList[PH_num].GetNextStationWithProcess(_MoverList[mv_i].Station));
                END_IF

            ApproachScenario_e.WaitOnFreeStation:
                IF NOT THIS^.GetPrevMover(_MoverList[mv_i]).Station.Equals(_MoverList[mv_i].Station) THEN
                    _MoverList[mv_i].MoveToStation();
                END_IF

            // wait on the previous station to be free (syncronize with the previous)
            ApproachScenario_e.WaitOnPrevProcess:
                // TODO implement !!!!
                _MoverList[mv_i].MoveToStation();

            // Move the mover only when all movers process are finished
            ApproachScenario_e.WaitOnExternalTrigger:
                IF bMoverSync THEN
                    // move only when there are no mover currently going to the station
                    IF NOT THIS^.IsMoverMovingToStation(mv_i) THEN
                        _MoverList[mv_i].MoveToStation();
                    END_IF
                END_IF

            END_CASE

        MoverState_e.WaitLeaveCurrentStation:
            IF NOT CONST.BIND_WITH_TRACK THEN
                _MoverList[mv_i].State := MoverState_e.MovingToStation;
            ELSE
                IF NOT gMoverAxis.I_CT_Shuttle_from_BR.asStruct[mv_i].bStatus.at_target THEN
                    _MoverList[mv_i].State := MoverState_e.MovingToStation;
                END_IF
            END_IF

        MoverState_e.MovingToStation:
            IF _MoverList[mv_i].IsInStationPos() THEN
                _MoverList[mv_i].State := MoverState_e.InStationPos;

            ELSIF NOT __ISVALIDREF(_MoverList[mv_i].Station) THEN
                ASSERT(0);
                _MoverList[mv_i].State := MoverState_e.WaitOnNextStation;
                _MoverList[mv_i].SetStation(_WorkStationList[PH_num].GetNextStation(_MoverList[mv_i].Station));

            ELSIF __ISVALIDREF(_MoverList[mv_i].Station.Process) AND NOT CONST.BIND_WITH_TRACK THEN
                iNumOfMoverOnTheWay := THIS^.GetNumOfMoverOnTheWay(_MoverList[mv_i]);

                IF _MoverList[mv_i].Station.Process.xMoverPathFree AND
                   NOT (_MoverList[mv_i].Station.Equals(THIS^.GetNextMover(_MoverList[mv_i]).Station)) AND
                   (iNumOfMoverOnTheWay <= _MoverList[mv_i].Station.iMaxWaitingMovers) THEN
                    _MoverList[mv_i].MoveToStation();
                END_IF

            ELSIF _MoverList[mv_i].MoverAxis.isInPos AND NOT CONST.BIND_WITH_TRACK THEN
                _MoverList[mv_i].MoveToStation();
            END_IF

        MoverState_e.InStationPos:
            IF NOT __ISVALIDREF(_MoverList[mv_i].Station) THEN
                ASSERT(0);
                _MoverList[mv_i].State := MoverState_e.WaitOnNextStation;
                _MoverList[mv_i].SetStation(_WorkStationList[PH_num].GetNextStation(_MoverList[mv_i].Station));

                // If there is no station (waiting position)
            ELSIF NOT __ISVALIDREF(_MoverList[mv_i].Station.Process) THEN
                _MoverList[mv_i].State := MoverState_e.WaitOnNextStation;
                _MoverList[mv_i].SetStation(_WorkStationList[PH_num].GetNextStation(_MoverList[mv_i].Station));

            ELSE
                IF __ISVALIDREF(_MoverList[mv_i].Station.Process.Mover) THEN
                    // ASSERT(0); TODO we have to find why we are here so often.

                    IF _MoverList[mv_i].Station.Process.xMoverShouldLeave THEN
                        _MoverList[mv_i].Station.Process.TakeMover();
                        ASSERT(0);

                    ELSE
                        _MoverList[mv_i].State := MoverState_e.OperationDone;
                    END_IF
                ELSE
                    _MoverList[mv_i].Station.Process.GiveMover(_MoverList[mv_i]);
                    _MoverList[mv_i].State := MoverState_e.InOperation;
                END_IF
            END_IF

        MoverState_e.InOperation:
            IF NOT __ISVALIDREF(_MoverList[mv_i].Station) THEN
                ASSERT(0);
                _MoverList[mv_i].State := MoverState_e.WaitOnNextStation;
                _MoverList[mv_i].SetStation(_WorkStationList[PH_num].GetNextStation(_MoverList[mv_i].Station));

            ELSIF NOT __ISVALIDREF(_MoverList[mv_i].Station.Process) THEN
                ASSERT(0);
                _MoverList[mv_i].State := MoverState_e.OperationDone;

            ELSIF _MoverList[mv_i].Station.Process.xMoverShouldLeave THEN
                _MoverList[mv_i].State := MoverState_e.OperationDone;

            ELSIF NOT __ISVALIDREF(_MoverList[mv_i].Station.Process.Mover) THEN
                ASSERT(0);
                _MoverList[mv_i].Station.Process.GiveMover(_MoverList[mv_i]);
            END_IF

        MoverState_e.PerformRelativeMove:
            IF NOT __ISVALIDREF(_MoverList[mv_i].Station) THEN
                ASSERT(0);
                _MoverList[mv_i].State := MoverState_e.WaitOnNextStation;
                _MoverList[mv_i].SetStation(_WorkStationList[PH_num].GetNextStation(_MoverList[mv_i].Station));

            ELSIF NOT __ISVALIDREF(_MoverList[mv_i].Station.Process) THEN
                ASSERT(0);
                _MoverList[mv_i].State := MoverState_e.OperationDone;

            ELSIF _MoverList[mv_i].Station.Process.xMoverShouldLeave THEN
                _MoverList[mv_i].State := MoverState_e.OperationDone;

            ELSE
                IF NOT _MoverList[mv_i].IsInStationPos() THEN
                    _MoverList[mv_i].State := MoverState_e.WaitRelativeMoveEnd;
                END_IF

            END_IF

        MoverState_e.WaitRelativeMoveEnd:
            IF NOT __ISVALIDREF(_MoverList[mv_i].Station) THEN
                ASSERT(0);
                _MoverList[mv_i].State := MoverState_e.WaitOnNextStation;
                _MoverList[mv_i].SetStation(_WorkStationList[PH_num].GetNextStation(_MoverList[mv_i].Station));

            ELSIF NOT __ISVALIDREF(_MoverList[mv_i].Station.Process) THEN
                ASSERT(0);
                _MoverList[mv_i].State := MoverState_e.OperationDone;

            ELSE
                IF _MoverList[mv_i].IsInStationPos() THEN
                    _MoverList[mv_i].State := MoverState_e.InOperation;

                ELSIF gMoverAxis.I_CT_Shuttle_from_BR.asStruct[mv_i].bStatus.at_target THEN
                    _MoverList[mv_i].State := MoverState_e.PerformRelativeMove;
                END_IF

            END_IF

        END_CASE
    END_IF
END_FOR

// update bMoverSync
bMoverSync := THIS^.IsAllMoverAtPosition() OR THIS^.IsMoverStucked();

